(* Logix 5000 project; controller CLASE_1 Emulate 5570 rev 28.11; software revision 28.02; part 9 of 15 *)
(* tags used below, declared in another part *)
   Inp_ActuatorFault : BOOL;   // Valve Actuator Fault (overload, etc.), 0=OK, 1=Fault)
   Cfg_SetTrack : BOOL;   // 1=PSets track OSets in Oper, OSets track PSets in Prog, 0=no tracking
   Cfg_SetTrackOvrdHand : BOOL;   // 1=Prog/Oper Settings track Override/Hand CV
   Cfg_MinCV : REAL;   // Minimum CV (in CV EU, for limiting)
   Cfg_MaxCV : REAL;   // Maximum CV (in CV EU, for limiting)
   Cfg_CycleT : REAL;   // Open and Close Pulse Output overall period (s)
   Cfg_OpenRate : REAL;   // Rate at which valve moves when opening (CV EU/sec)
   Cfg_CloseRate : REAL;   // Rate at which valve moves when closing (CV EU/sec)
   Cfg_MaxOnT : REAL;   // Open and Close Pulse Output maximum ON time (s)
   Cfg_MinOnT : REAL;   // Open and Close Pulse Output minimum ON time (s)
   Cfg_BumpT : REAL;   // Time to bump valve open or closed (by Oper) when Fdbk Bad (sec)
   Cfg_Deadtime : REAL;   // Additional time on first pulse after stop or direction change
   PSet_CV : REAL;   // Program Setting of Controlled Variable (output) (CV EU)
   PSet_CVRoCLimInc : REAL;   // Program Setting of CV Rate of Change Limit, Increasing, (in EU/sec)
   PSet_CVRoCLimDec : REAL;   // Program Setting of CV Rate of Change Limit, Decreasing, (in EU/sec)
   OSet_CV : REAL;   // Operator Setting of Controlled Variable (output) (CV EU)
   OSet_CVRoCLimInc : REAL;   // Operator Setting of CV Rate of Change Limit, Increasing, (in EU/sec)
   OSet_CVRoCLimDec : REAL;   // Operator Setting of CV Rate of Change Limit, Decreasing, (in EU/sec)
   Out_Open : BOOL;   // Pulse Output to drive valve Open
   Out_Close : BOOL;   // Pulse Output to drive valve closed
   Val_Pos : REAL;   // Valve actual position from feedback (CV EU)
   Val_CVSet : REAL;   // Value of selected CV Setting (before rate limiting, CV EU)
   Val_CVOut : REAL;   // Value of CV output (after clamping and ramping) (CV EU)
   Val_CVRoCLimInc : REAL;   // Value of CV Rate of Change Limit, Increasing, (in EU/sec)
   Val_CVRoCLimDec : REAL;   // Value of CV Rate of Change Limit, Decreasing, (in EU/sec)
   Sts_BumpOpen : BOOL;   // 1=Bump Open Requested or Active
   Sts_BumpClose : BOOL;   // 1=Bump Close Requested or Active
   Sts_Ramping : BOOL;   // 1=CV is ramping to target
   Sts_Clamped : BOOL;   // 1=CV Set is clamped at CVMin or CVMax
   P_ValveC : BOOL;   // Unique Parameter Name for auto - discovery
   Wrk_CVRoCLimInc : REAL;   // Selected CV Rate of Change Limit Increasing
   Wrk_CVSet : REAL;   // Final selected CV to feed to RoC Limiter
   Wrk_CVOut : REAL;   // Working value of CV after Rate Limiting
   ActuatorFault : P_Alarm;   // Actuator Fault Alarm (based on Actuator Fault Input)
   Wrk_Close : BOOL;   // Internal Close output -- before Sim
   Wrk_CycleT : TIMER;   // Overall Cycle Timer for pulsed outputs
   Wrk_OKtoOpen : BOOL;   // OK to pulse Out_Open
   Wrk_OKtoClose : BOOL;   // OK to pulse Out_Close
   Wrk_OpenTime : REAL;   // Time to pulse Out_Open
   Wrk_CycleT_ms : DINT;   // Cycle Time in milliseconds (preset)
   Wrk_OpenTimePrev : DINT;   // Wrk_OpenTime from previous cycle
   Wrk_CloseTime : REAL;   // Time to pulse Out_Close
   Wrk_CloseTimePrev : REAL;   // Wrk_CloseTime from previous cycle
   Wrk_CVRoCLimDec : REAL;   // Selected CV Rate of Change Limit Decreasing
   Wrk_BumpClose : BOOL;   // Operator Bump Close requested
   Wrk_BumpOpen : BOOL;   // Operator Bump Open requested
   Wrk_BumpingOpen : BOOL;   // Operator Bump Open actively pulsing Out_Open
   Wrk_BumpingClose : BOOL;   // Operator Bump Close actively pulsing Out_Close
   Wrk_CycleActive : BOOL;   // Outputs are cycling; wait for cycle to complete
   Wrk_ShedIntlkCV : BOOL;   // Output CV being held at Interlock value
   Wrk_ShedHold : BOOL;   // Output CV being held at last good value
(* P_ValveC, continued *)

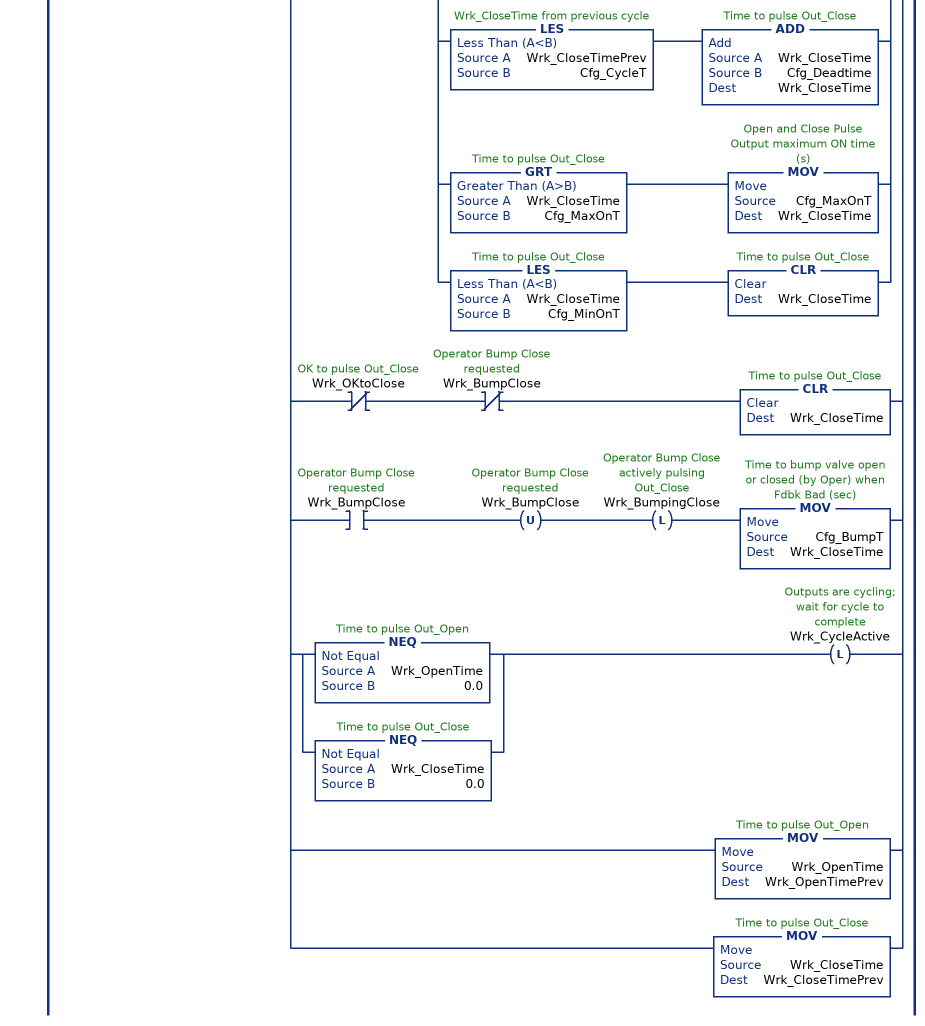
   // When the Cycle completes, calculate a new Open Time (time to pulse the
   // Open output) and Close Time (time to pulse the Close output).
   // Details of this calculation are in the Instruction Help for the POSP built-in
   // instruction, from which this logic is derived.
   48: [GEQ(Wrk_CycleT.ACC,Wrk_CycleT_ms) ,XIO(Wrk_CycleActive) ][OTU(Wrk_CycleActive) OTU(Wrk_BumpingOpen) OTU(Wrk_BumpingClose) CLR(Wrk_CycleT.ACC) ,XIC(Wrk_OKtoOpen) [CPT(Wrk_OpenTime,(Val_CVOut-Val_Pos)/Cfg_OpenRate) ,LES(Wrk_OpenTimePrev,Cfg_CycleT) ADD(Wrk_OpenTime,Cfg_Deadtime,Wrk_OpenTime) ,GRT(Wrk_OpenTime,Cfg_MaxOnT) MOV(Cfg_MaxOnT,Wrk_OpenTime) ,LES(Wrk_OpenTime,Cfg_MinOnT) CLR(Wrk_OpenTime) ] ,XIO(Wrk_OKtoOpen) XIO(Wrk_BumpOpen) CLR(Wrk_OpenTime) ,XIC(Wrk_BumpOpen) OTU(Wrk_BumpOpen) OTL(Wrk_BumpingOpen) MOV(Cfg_BumpT,Wrk_OpenTime) ,XIC(Wrk_OKtoClose) [CPT(Wrk_CloseTime,(Val_Pos-Val_CVOut)/Cfg_CloseRate) ,LES(Wrk_CloseTimePrev,Cfg_CycleT) ADD(Wrk_CloseTime,Cfg_Deadtime,Wrk_CloseTime) ,GRT(Wrk_CloseTime,Cfg_MaxOnT) MOV(Cfg_MaxOnT,Wrk_CloseTime) ,LES(Wrk_CloseTime,Cfg_MinOnT) CLR(Wrk_CloseTime) ] ,XIO(Wrk_OKtoClose) XIO(Wrk_BumpClose) CLR(Wrk_CloseTime) ,XIC(Wrk_BumpClose) OTU(Wrk_BumpClose) OTL(Wrk_BumpingClose) MOV(Cfg_BumpT,Wrk_CloseTime) ,[NEQ(Wrk_OpenTime,0.0) ,NEQ(Wrk_CloseTime,0.0) ] OTL(Wrk_CycleActive) ,MOV(Wrk_OpenTime,Wrk_OpenTimePrev) ,MOV(Wrk_CloseTime,Wrk_CloseTimePrev) ];
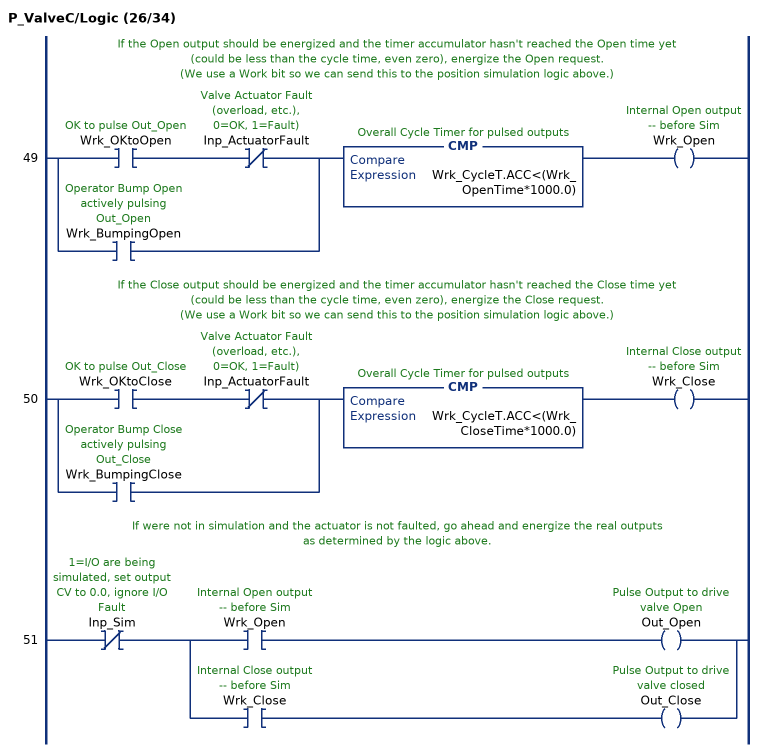
   // If the Open output should be energized and the timer accumulator hasn't reached the Open time yet
   // (could be less than the cycle time, even zero), energize the Open request.
   // (We use a Work bit so we can send this to the position simulation logic above.)
   49: [XIC(Wrk_OKtoOpen) XIO(Inp_ActuatorFault) ,XIC(Wrk_BumpingOpen) ]CMP(Wrk_CycleT.ACC<(Wrk_OpenTime*1000.0))OTE(Wrk_Open);
   // If the Close output should be energized and the timer accumulator hasn't reached the Close time yet
   // (could be less than the cycle time, even zero), energize the Close request.
   // (We use a Work bit so we can send this to the position simulation logic above.)
   50: [XIC(Wrk_OKtoClose) XIO(Inp_ActuatorFault) ,XIC(Wrk_BumpingClose) ]CMP(Wrk_CycleT.ACC<(Wrk_CloseTime*1000.0))OTE(Wrk_Close);
   // If were not in simulation and the actuator is not faulted, go ahead and energize the real outputs
   // as determined by the logic above.
   51: XIO(Inp_Sim)[XIC(Wrk_Open) OTE(Out_Open) ,XIC(Wrk_Close) OTE(Out_Close) ];
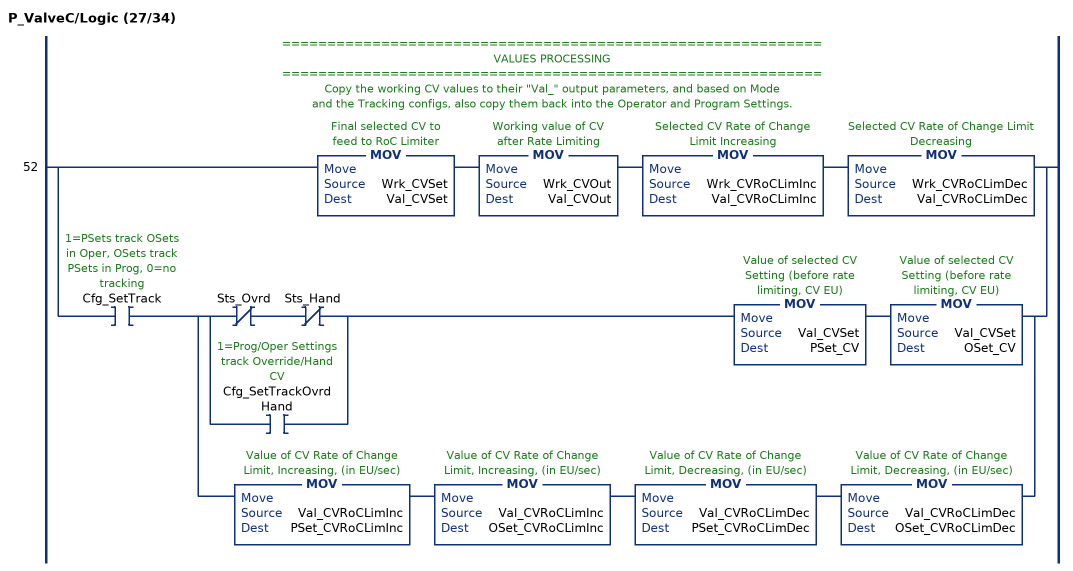
   // ============================================================
   // VALUES PROCESSING
   // ============================================================
   // Copy the working CV values to their "Val_" output parameters, and based on Mode
   // and the Tracking configs, also copy them back into the Operator and Program Settings.
   52: [MOV(Wrk_CVSet,Val_CVSet) MOV(Wrk_CVOut,Val_CVOut) MOV(Wrk_CVRoCLimInc,Val_CVRoCLimInc) MOV(Wrk_CVRoCLimDec,Val_CVRoCLimDec) ,XIC(Cfg_SetTrack) [[XIO(Sts_Ovrd) XIO(Sts_Hand) ,XIC(Cfg_SetTrackOvrdHand) ] MOV(Val_CVSet,PSet_CV) MOV(Val_CVSet,OSet_CV) ,MOV(Val_CVRoCLimInc,PSet_CVRoCLimInc) MOV(Val_CVRoCLimInc,OSet_CVRoCLimInc) MOV(Val_CVRoCLimDec,PSet_CVRoCLimDec) MOV(Val_CVRoCLimDec,OSet_CVRoCLimDec) ] ];
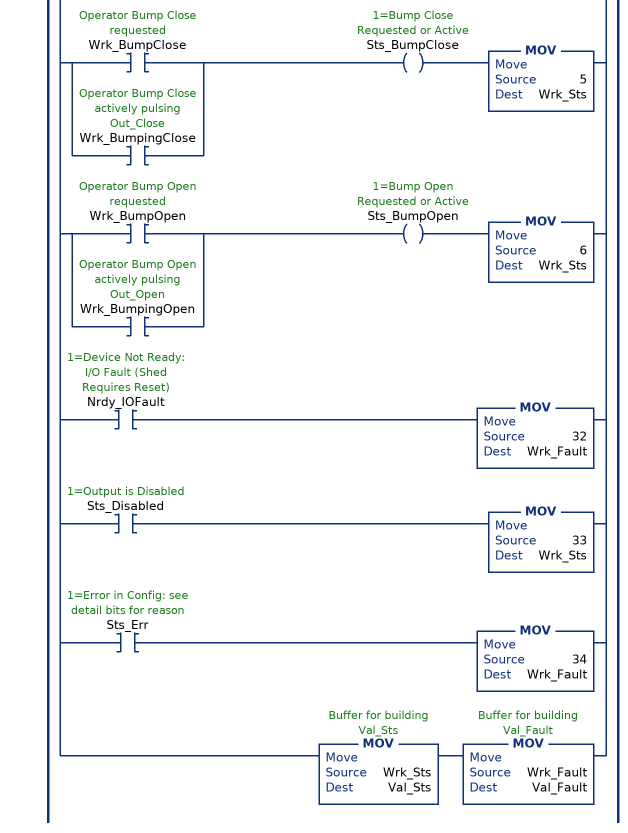
   // Val_Sts is the current device status, as determined by this AOI,
   // based on its knowledge of settings and configuration.
   // (This is the status that should be monitored by, for example, FT Historian.)
   // 0 = At Target
   // 1 = Ramping Down
   // 2 = Ramping Up
   // 3 = Clamped at CVMin
   // 4 = Clamped at CVMax
   // 5 = Bump Close requested or currently pulsing Out_Close
   // 6 = Bump Open requested or currently pulsing Out_Open
   // 32 = I/O Fault
   // 33 = Disabled
   // 34 = Configuration Error
   // #####  V3.0-04  2014-01-20:  Corrected generation of Val_Sts, Val_Fault.  #####
   // #####  V3.1-00  2014-07-22: Added Not Ready reason bits (Nrdy_xxx)  #####
   // #####  V3.1-03  2015-01-21:  Modified to show Val_Sts = 1 or 2 when moving via pulsing.  #####
   53: [CLR(Wrk_Sts) CLR(Wrk_Fault) ,[GRT(Wrk_OpenTime,0.0) XIO(Inp_ActuatorFault) ,XIC(Sts_Ramping) LES(Wrk_CVOut,Wrk_CVSet) ] MOV(2,Wrk_Sts) ,[GRT(Wrk_CloseTime,0.0) XIO(Inp_ActuatorFault) ,XIC(Sts_Ramping) GRT(Wrk_CVOut,Wrk_CVSet) ] MOV(1,Wrk_Sts) ,XIC(Sts_Clamped) [EQU(Wrk_CVOut,Cfg_MinCV) MOV(3,Wrk_Sts) ,EQU(Wrk_CVOut,Cfg_MaxCV) MOV(4,Wrk_Sts) ] ,[XIC(Wrk_BumpClose) ,XIC(Wrk_BumpingClose) ] OTE(Sts_BumpClose) MOV(5,Wrk_Sts) ,[XIC(Wrk_BumpOpen) ,XIC(Wrk_BumpingOpen) ] OTE(Sts_BumpOpen) MOV(6,Wrk_Sts) ,XIC(Nrdy_IOFault) MOV(32,Wrk_Fault) ,XIC(Sts_Disabled) MOV(33,Wrk_Sts) ,XIC(Sts_Err) MOV(34,Wrk_Fault) ,MOV(Wrk_Sts,Val_Sts) MOV(Wrk_Fault,Val_Fault) ];
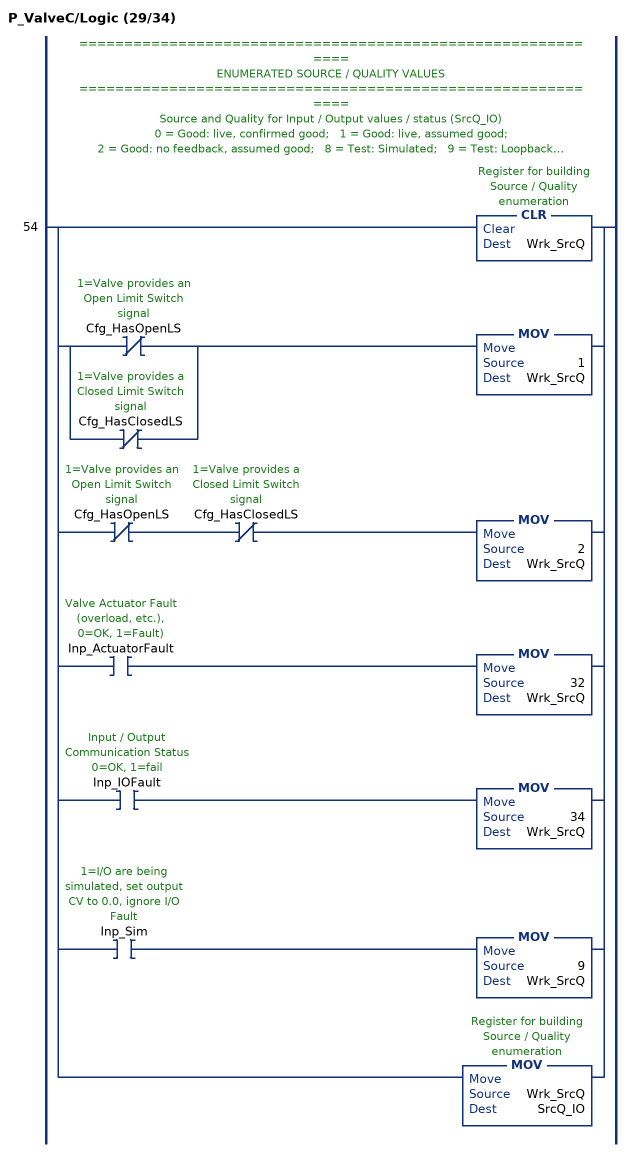
   // ============================================================
   // ENUMERATED SOURCE / QUALITY VALUES
   // ============================================================
   // Source and Quality for Input / Output values / status (SrcQ_IO)
   // 0 = Good: live, confirmed good;   1 = Good: live, assumed good;
   // 2 = Good: no feedback, assumed good;   8 = Test: Simulated;   9 = Test: Loopback;
   // 10 = Test: Manually Entered;   16 = Uncertain: Live, off-spec;
   // 17 = Uncertain, Substituted at Device / Bus;   18 = Uncertain, Substituted at AOI;
   // 19 = Uncertain, using last known good;    20 = Uncertain, using replacement value;
   // 32 = Bad, Signal Failure;   33 = Bad, Channel Fault;
   // 34 = Bad, Module / Comms Fault;   35 = Bad, Invalid Configuration
   // #####  V3.1-00  2014-07-22:  Added rung for Source/Quality enumerations.  #####
   54: [CLR(Wrk_SrcQ) ,[XIO(Cfg_HasOpenLS) ,XIO(Cfg_HasClosedLS) ] MOV(1,Wrk_SrcQ) ,XIO(Cfg_HasOpenLS) XIO(Cfg_HasClosedLS) MOV(2,Wrk_SrcQ) ,XIC(Inp_ActuatorFault) MOV(32,Wrk_SrcQ) ,XIC(Inp_IOFault) MOV(34,Wrk_SrcQ) ,XIC(Inp_Sim) MOV(9,Wrk_SrcQ) ,MOV(Wrk_SrcQ,SrcQ_IO) ];
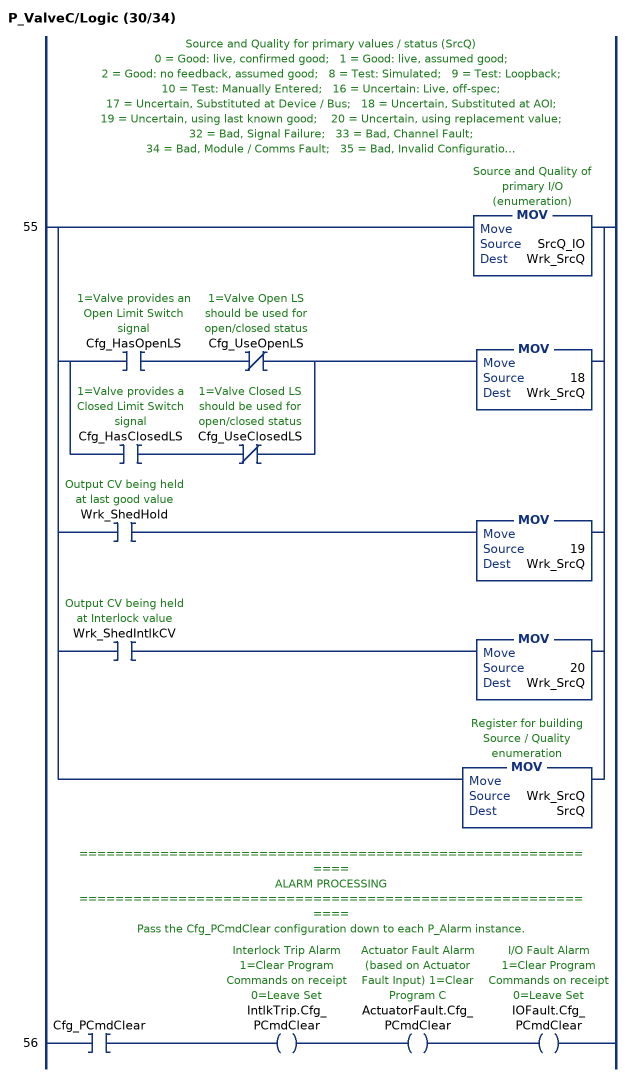
   // Source and Quality for primary values / status (SrcQ)
   // 0 = Good: live, confirmed good;   1 = Good: live, assumed good;
   // 2 = Good: no feedback, assumed good;   8 = Test: Simulated;   9 = Test: Loopback;
   // 10 = Test: Manually Entered;   16 = Uncertain: Live, off-spec;
   // 17 = Uncertain, Substituted at Device / Bus;   18 = Uncertain, Substituted at AOI;
   // 19 = Uncertain, using last known good;    20 = Uncertain, using replacement value;
   // 32 = Bad, Signal Failure;   33 = Bad, Channel Fault;
   // 34 = Bad, Module / Comms Fault;   35 = Bad, Invalid Configuration
   // #####  V3.1-00  2014-07-22:  Added rung for Source/Quality enumerations.  #####
   55: [MOV(SrcQ_IO,Wrk_SrcQ) ,[XIC(Cfg_HasOpenLS) XIO(Cfg_UseOpenLS) ,XIC(Cfg_HasClosedLS) XIO(Cfg_UseClosedLS) ] MOV(18,Wrk_SrcQ) ,XIC(Wrk_ShedHold) MOV(19,Wrk_SrcQ) ,XIC(Wrk_ShedIntlkCV) MOV(20,Wrk_SrcQ) ,MOV(Wrk_SrcQ,SrcQ) ];
   // ============================================================
   // ALARM PROCESSING
   // ============================================================
   // Pass the Cfg_PCmdClear configuration down to each P_Alarm instance.
   56: XIC(Cfg_PCmdClear)OTE(IntlkTrip.Cfg_PCmdClear)OTE(ActuatorFault.Cfg_PCmdClear)OTE(IOFault.Cfg_PCmdClear);
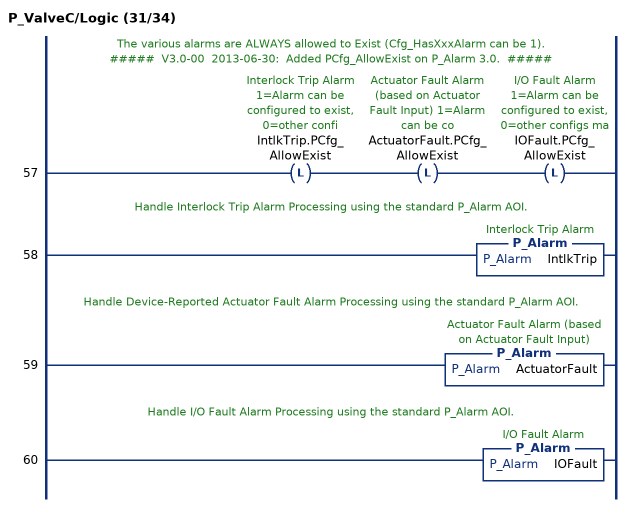
   // The various alarms are ALWAYS allowed to Exist (Cfg_HasXxxAlarm can be 1).
   // #####  V3.0-00  2013-06-30:  Added PCfg_AllowExist on P_Alarm 3.0.  #####
   57: OTL(IntlkTrip.PCfg_AllowExist)OTL(ActuatorFault.PCfg_AllowExist)OTL(IOFault.PCfg_AllowExist);
   // Handle Interlock Trip Alarm Processing using the standard P_Alarm AOI.
   58: P_Alarm(IntlkTrip);
   // Handle Device-Reported Actuator Fault Alarm Processing using the standard P_Alarm AOI.
   59: P_Alarm(ActuatorFault);
   // Handle I/O Fault Alarm Processing using the standard P_Alarm AOI.
   60: P_Alarm(IOFault);
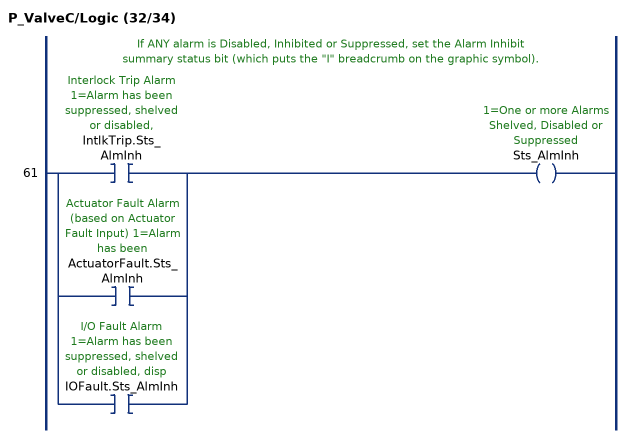
   // If ANY alarm is Disabled, Inhibited or Suppressed, set the Alarm Inhibit
   // summary status bit (which puts the "I" breadcrumb on the graphic symbol).
   61: [XIC(IntlkTrip.Sts_AlmInh) ,XIC(ActuatorFault.Sts_AlmInh) ,XIC(IOFault.Sts_AlmInh) ]OTE(Sts_AlmInh);
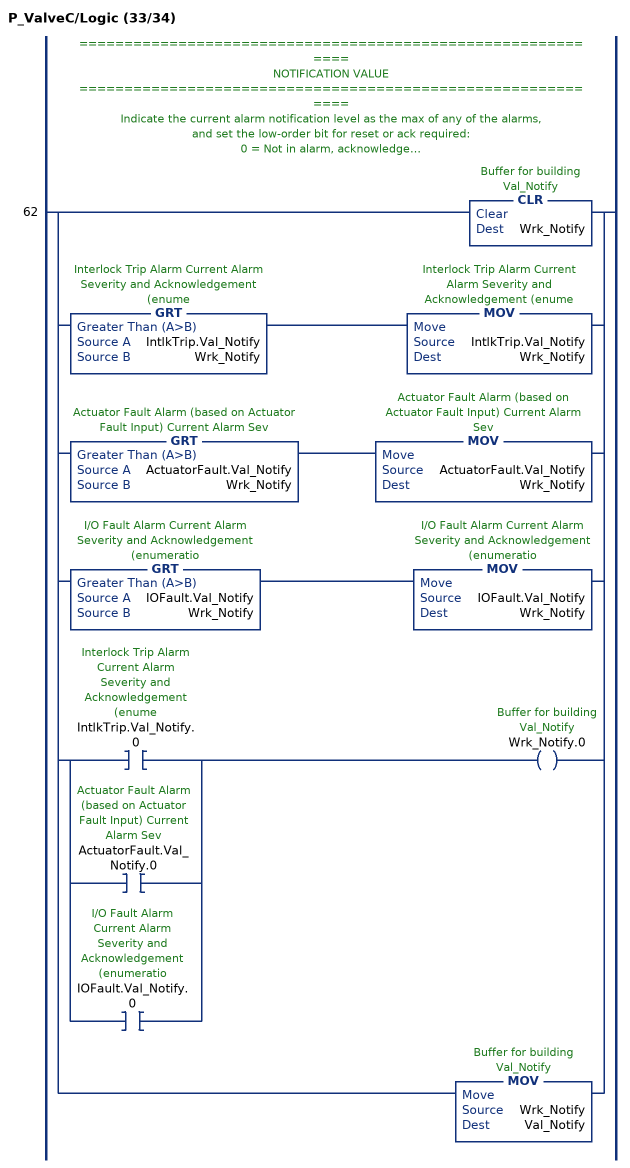
   // ============================================================
   // NOTIFICATION VALUE
   // ============================================================
   // Indicate the current alarm notification level as the max of any of the alarms,
   // and set the low-order bit for reset or ack required:
   // 0 = Not in alarm, acknowledged
   // 1 = Not in alarm, unacknowledged or reset required
   // 2 = Low severity alarm, acknowledged
   // 3 = Low severity alarm, unacknowledged
   // 4 = Medium severity alarm, acknowledged
   // 5 = Medium severity alarm, unacknowledged
   // 6 = High severity alarm, acknowledged
   // 7 = High severity alarm, unacknowledged
   // 8 = Urgent severity alarm, acknowledged
   // 9 = Urgent severity alarm, unacknowledged
   // #####  V3.1-00  2014-07-22:  Separated Reset Reqd functions from Val_Notify  #####
   62: [CLR(Wrk_Notify) ,GRT(IntlkTrip.Val_Notify,Wrk_Notify) MOV(IntlkTrip.Val_Notify,Wrk_Notify) ,GRT(ActuatorFault.Val_Notify,Wrk_Notify) MOV(ActuatorFault.Val_Notify,Wrk_Notify) ,GRT(IOFault.Val_Notify,Wrk_Notify) MOV(IOFault.Val_Notify,Wrk_Notify) ,[XIC(IntlkTrip.Val_Notify.0) ,XIC(ActuatorFault.Val_Notify.0) ,XIC(IOFault.Val_Notify.0) ] OTE(Wrk_Notify.0) ,MOV(Wrk_Notify,Val_Notify) ];
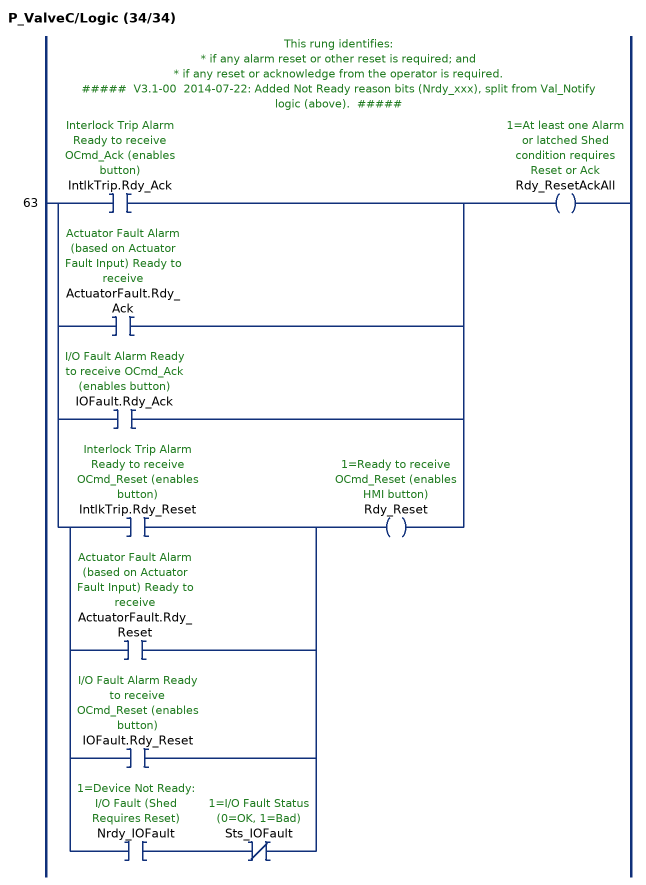
   // This rung identifies:
   // * if any alarm reset or other reset is required; and
   // * if any reset or acknowledge from the operator is required.
   // #####  V3.1-00  2014-07-22: Added Not Ready reason bits (Nrdy_xxx), split from Val_Notify logic (above).  #####
   63: [[XIC(IntlkTrip.Rdy_Ack) ,XIC(ActuatorFault.Rdy_Ack) ,XIC(IOFault.Rdy_Ack) ] ,[XIC(IntlkTrip.Rdy_Reset) ,XIC(ActuatorFault.Rdy_Reset) ,XIC(IOFault.Rdy_Reset) ,XIC(Nrdy_IOFault) XIO(Sts_IOFault) ] OTE(Rdy_Reset) ]OTE(Rdy_ResetAckAll);
END_ROUTINE

ROUTINE Prescan   (* ladder *)
// Clear Ownership. clear "lurking" Commands
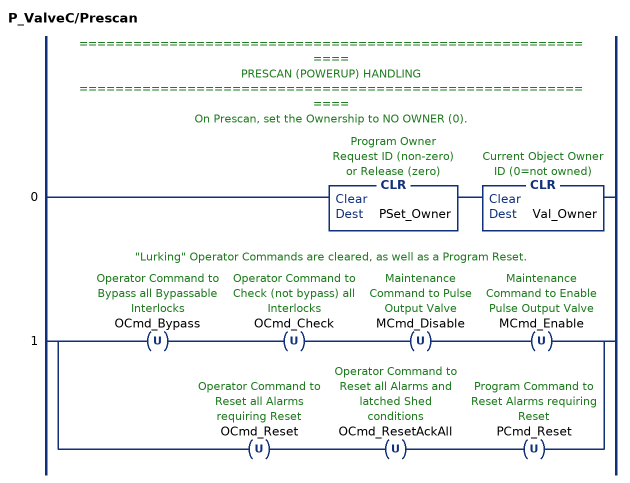
   // ============================================================
   // PRESCAN (POWERUP) HANDLING
   // ============================================================
   // On Prescan, set the Ownership to NO OWNER (0).
   0: CLR(PSet_Owner)CLR(Val_Owner);
   // "Lurking" Operator Commands are cleared, as well as a Program Reset.
   1: [OTU(OCmd_Bypass) OTU(OCmd_Check) OTU(MCmd_Disable) OTU(MCmd_Enable) ,OTU(OCmd_Reset) OTU(OCmd_ResetAckAll) OTU(PCmd_Reset) ];
END_ROUTINE
END_ADD_ON_INSTRUCTION

ADD_ON_INSTRUCTION P_ValveSO   (* revision 3.5 04 Release, vendor Rockwell Automation, ExecutePrescan, ExecuteEnableInFalse *)
// Solenoid Operated Valve
// Revision note:
// See V3.5-xx Release Notes for details. Modified to align
// with actual device state on transition from Sim to real valve.
// Help:
// Copyright © Rockwell Automation, Inc.  All Rights Reserved.
// This Instruction controls and monitors a single solenoid operated
// valve (two position: opened, closed) and provides:
// *  Support for fail open (energize to close) and fail closed (energize to open, default) valves
// *  Monitoring of limit switch feedback, display of actual valve status
// *  Detection of Failure to Open, Failure to Close
// *  Monitoring of Permissive conditions to allow energizing
// *  Monitoring of Interlock conditions to de-energize
// *  Simulation, providing feedback of a working valve while disabling outputs
// *  Monitoring of I/O communication faults
// *  Alarms for Full Stall (didn't move), Transit Stall (didn't reach target position), Interlock Trip, I/O Fault
// *  Operation in Hand, Maintenance, Override, Program and Operator Modes
// *  "Available" status for use by automation logic to know whether valve
//       can be controlled by other objects.
// Modes are provided by a P_Mode AOI instance.
// Alarms are provided by P_Alarm AOI instances.
// Modes of operation: Operator, Program, Override, Maintenance, Hand
VAR_INPUT
   Inp_OpenLS : BOOL; {visible}   // Valve Open Limit Switch 1=confirmed OPEN
   Inp_ClosedLS : BOOL; {visible}   // Valve Closed Limit Switch 1=confirmed CLOSED
   Inp_PermOK : BOOL := 1; {visible}   // 1=Permissives OK, Valve can energize
   Inp_NBPermOK : BOOL := 1; {visible}   // 1=Non-Bypassable Permissives OK, valve can energize
   Inp_IntlkOK : BOOL := 1; {visible}   // 1=Interlocks OK, valve can energize
   Inp_NBIntlkOK : BOOL := 1; {visible}   // 1=Non-Bypassable Interlocks OK, valve can energize
   Inp_IOFault : BOOL;   // Input Communication Status 0=OK, 1=fail
   Inp_Sim : BOOL;   // 1=Simulate working valve; 0=Open/Close/ Monitor actual valve
   Inp_Hand : ALIAS FOR Mode.Inp_Hand; {visible}
   Inp_Ovrd : ALIAS FOR Mode.Inp_Ovrd; {visible}
   Inp_OvrdCmd : DINT; {visible}   // Override Mode Command: 0=None, 1=Close, 2=Open
   Inp_Reset : BOOL; {visible}   // 1=Reset all fault conditions and latched Alarms
   Cfg_FailOpen : BOOL;   // 1=Fail Open (energize to close), 0=Fail Closed (energize to open)
   Cfg_HasOpenLS : BOOL;   // 1=Valve provides an Open Limit Switch signal
   Cfg_HasClosedLS : BOOL;   // 1=Valve provides a Closed Limit Switch signal
   Cfg_UseOpenLS : BOOL;   // 1=Valve Open LS should be used for failure checking
   Cfg_UseClosedLS : BOOL;   // 1=Valve Closed LS should be used for failure checking
   Cfg_LSFail : BOOL := 1;   // 1=both switches ON=fail, 0=both switches OFF=fail
   Cfg_HasPermObj : BOOL;   // 1=Tells HMI a P_Perm is connected to Inp_Perm
   Cfg_HasIntlkObj : BOOL;   // 1=Tells HMI a P_Intlk is connected to Inp_Intlk
   Cfg_HasStatsObj : BOOL;   // 1=Tells HMI a P_ValveStats is monitoring this valve
   Cfg_PCmdClear : ALIAS FOR Mode.Cfg_PCmdClear;
   Cfg_ProgDefault : ALIAS FOR Mode.Cfg_ProgDefault;
   Cfg_OCmdResets : BOOL;   // 1=New Oper valve cmd. resets fault, 0=reset req'd to clear fault
   Cfg_ShedOnFullStall : BOOL := 1;   // 1=Stop Valve and Alarm on Full Stall; 0=Alarm only on Full Stall
   Cfg_ShedOnTransitStall : BOOL := 1;   // 1=Stop Valve and Alarm on Transit Stall; 0=Alarm only on Transit Stall
   Cfg_ShedOnIOFault : BOOL := 1;   // 1=Stop Valve and Alarm on I/O Fault; 0=Alarm only on I/O Fault
   Cfg_OvrdPermIntlk : BOOL;   // 1=Override ignores Bypassable Perm/ Intlk; 0=always use Perm/Intlk
   Cfg_HasFullStallAlm : ALIAS FOR FullStall.Cfg_Exists;   // 1=Full Stall Alarm exists and will be checked
   Cfg_HasTransitStallAlm : ALIAS FOR TransitStall.Cfg_Exists;   // 1=Transit Stall Alarm exists and will be checked
   Cfg_HasIntlkTripAlm : ALIAS FOR IntlkTrip.Cfg_Exists;   // 1=Interlock Trip Alarm exists and will be checked
   Cfg_HasIOFaultAlm : ALIAS FOR IOFault.Cfg_Exists;   // 1=I/O Fault Alarm exists and will be checked
   Cfg_FullStallResetReqd : ALIAS FOR FullStall.Cfg_ResetReqd;   // 1=Reset requied to clear Full Stall Alarm
   Cfg_TransitStallResetReqd : ALIAS FOR TransitStall.Cfg_ResetReqd;   // 1=Reset required to clear Transit Stall Alarm
   Cfg_IntlkTripResetReqd : ALIAS FOR IntlkTrip.Cfg_ResetReqd;   // 1=Reset required to clear Interlock Trip Alarm
   Cfg_IOFaultResetReqd : ALIAS FOR IOFault.Cfg_ResetReqd;   // 1=Reset required to clear I/O Fault Alarm
   Cfg_FullStallAckReqd : ALIAS FOR FullStall.Cfg_AckReqd;   // 1=Acknowledge required for Full Stall Alarm
   Cfg_TransitStallAckReqd : ALIAS FOR TransitStall.Cfg_AckReqd;   // 1=Acknowledge required for Transit Stall Alarm
   Cfg_IntlkTripAckReqd : ALIAS FOR IntlkTrip.Cfg_AckReqd;   // 1=Acknowledge required for Interlock Trip Alarm
   Cfg_IOFaultAckReqd : ALIAS FOR IOFault.Cfg_AckReqd;   // 1=Acknowledge required for I/O Fault Alarm
   Cfg_FullStallSeverity : ALIAS FOR FullStall.Cfg_Severity;   // Full Stall Alarm Severity: 1..250=Low, 251..500=Medium, 501..750=High, 751..1000=Urgent
   Cfg_TransitStallSeverity : ALIAS FOR TransitStall.Cfg_Severity;   // Transit Stall Alarm Severity: 1..250=Low, 251..500=Medium, 501..750=High, 751..1000=Urgent
   Cfg_IntlkTripSeverity : ALIAS FOR IntlkTrip.Cfg_Severity;   // Interlock Trip Alarm Severity: 1..250=Low, 251..500=Medium, 501..750=High, 751..1000=Urgent
   Cfg_IOFaultSeverity : ALIAS FOR IOFault.Cfg_Severity;   // I/O Fault Alarm Severity: 1..250=Low, 251..500=Medium, 501..750=High, 751..1000=Urgent
   Cfg_SimFdbkT : DINT := 2;   // Delay to echo back of Open/Closed status when in Simulation (sec)
   Cfg_FullStallT : DINT := 5;   // After command, time with no motion before Fault (sec)
   Cfg_TransitStallT : DINT := 10;   // After command, time to reach position before fault (sec)
   PSet_Owner : DINT;   // Program Owner Request ID (non-zero) or Release (zero)
   PCmd_Open : BOOL;   // Program Command to Open Valve
   PCmd_Close : BOOL;   // Program Command to Close Valve
   PCmd_Acq : ALIAS FOR Mode.PCmd_Acq;
   PCmd_Rel : ALIAS FOR Mode.PCmd_Rel;
   PCmd_Lock : ALIAS FOR Mode.PCmd_Lock;
   PCmd_Unlock : ALIAS FOR Mode.PCmd_Unlock;
   PCmd_Reset : BOOL;   // Program Command to Reset all Alarms requiring Reset
   PCmd_FullStallAck : ALIAS FOR FullStall.PCmd_Ack;   // Program Command to Acknowledge Full Stall Alarm
   PCmd_FullStallSuppress : ALIAS FOR FullStall.PCmd_Suppress;   // Program Command to Suppress Full Stall Alarm
   PCmd_FullStallUnsuppress : ALIAS FOR FullStall.PCmd_Unsuppress;   // Program Command to Unsuppress Full Stall Alarm
   PCmd_FullStallUnshelve : ALIAS FOR FullStall.PCmd_Unshelve;   // Program Command to Unshelve Full Stall Alarm
   PCmd_TransitStallAck : ALIAS FOR TransitStall.PCmd_Ack;   // Program Command to Acknowledge Transit Stall Alarm
   PCmd_TransitStallSuppress : ALIAS FOR TransitStall.PCmd_Suppress;   // Program Command to Suppress Transit Stall Alarm
   PCmd_TransitStallUnsuppress : ALIAS FOR TransitStall.PCmd_Unsuppress;   // Program Command to Unsuppress Transit Stall Alarm
   PCmd_TransitStallUnshelve : ALIAS FOR TransitStall.PCmd_Unshelve;   // Program Command to Unshelve Transit Stall Alarm
   PCmd_IntlkTripAck : ALIAS FOR IntlkTrip.PCmd_Ack;   // Program Command to Acknowledge Interlock Trip Alarm
   PCmd_IntlkTripSuppress : ALIAS FOR IntlkTrip.PCmd_Suppress;   // Program Command to Suppress Interlock Trip Alarm
   PCmd_IntlkTripUnsuppress : ALIAS FOR IntlkTrip.PCmd_Unsuppress;   // Program Command to Unsuppress Interlock Trip Alarm
   PCmd_IntlkTripUnshelve : ALIAS FOR IntlkTrip.PCmd_Unshelve;   // Program Command to Unshelve Interlock Trip Alarm
   PCmd_IOFaultAck : ALIAS FOR IOFault.PCmd_Ack;   // Program Command to Acknowledge I/O Fault Alarm
   PCmd_IOFaultSuppress : ALIAS FOR IOFault.PCmd_Suppress;   // Program Command to Suppress I/O Fault Alarm
   PCmd_IOFaultUnsuppress : ALIAS FOR IOFault.PCmd_Unsuppress;   // Program Command to Unsuppress I/O Fault Alarm
   PCmd_IOFaultUnshelve : ALIAS FOR IOFault.PCmd_Unshelve;   // Program Command to Unshelve I/O Fault Alarm
   OCmd_Open : BOOL;   // Operator Command to Open Valve
   OCmd_Close : BOOL;   // Operator Command to Close Valve
   OCmd_Bypass : BOOL;   // Operator Command to Bypass all Bypassable Interlocks and Permissives
   OCmd_Check : BOOL;   // Operator Command to Check (not bypass) all Interlocks and Permissives
   MCmd_Disable : BOOL;   // Maintenance Command to Disable Valve
   MCmd_Enable : BOOL;   // Maintenance Command to Enable (allow to energize) Valve
   MCmd_Acq : ALIAS FOR Mode.MCmd_Acq;
   MCmd_Rel : ALIAS FOR Mode.MCmd_Rel;
   OCmd_AcqLock : ALIAS FOR Mode.OCmd_AcqLock;
   OCmd_Unlock : ALIAS FOR Mode.OCmd_UnlockRel;
   OCmd_Reset : BOOL;   // Operator Command to Reset all Alarms requiring Reset
   OCmd_ResetAckAll : BOOL;   // Operator Command to Reset all Alarms and latched Shed conditions
END_VAR
VAR_OUTPUT
   Out : BOOL; {access Read Only, visible}   // 1=Energize Valve Solenoid
   SrcQ_IO : SINT; {access Read Only}   // Source and Quality of primary I/O (enumeration)
   SrcQ : SINT; {access Read Only}   // Source and Quality of primary Val/Sts (enumeration)
   Val_Cmd : SINT; {access Read Only}   // Device Command 0=None, 1=Close, 2=Open
   Val_Fdbk : SINT; {access Read Only}   // Device Feedback 0=Moving, 1=Closed, 2=Opened, 3=Limit Switch Failure
   Val_Sts : SINT; {access Read Only}   // Device Confirmed Sts 0=? 1=Closed 2=Open 5=Closing, 6=Opening, 33=Disabled
   Val_Fault : SINT; {access Read Only}   // Device Fault Status 0=None, 16=Transit Stall, 17 = Full Stall, 32=I/O Fault, 34=Config Error
   Val_Mode : ALIAS FOR Mode.Val; {access Read Only}
   Val_Owner : DINT; {access Read Only}   // Current Object Owner ID (0=not owned)
   Val_Notify : SINT; {access Read Only}   // Current Alarm Level and Acknowledgement (enumeration)
   Sts_Closed : BOOL; {access Read Only, visible}   // 1=Valve requested to Close and is confirmed Closed
   Sts_Opening : BOOL; {access Read Only, visible}   // 1=Valve requested to open and awaiting open feedback
   Sts_Opened : BOOL; {access Read Only, visible}   // 1=Valve requested to open and is confirmed Opened
   Sts_Closing : BOOL; {access Read Only, visible}   // 1=Valve requested to Close and awaiting Closed feedback
   Sts_Available : BOOL; {access Read Only}   // 1=Valve available for control by automation (Prog)
   Sts_Bypass : BOOL; {access Read Only}   // 1=Bypassable Interlocks and Permissives are Bypassed
   Sts_BypActive : BOOL; {access Read Only}   // 1=Bypassing Active (Bypassed or Maintenance)
   Sts_Disabled : BOOL; {access Read Only}   // 1=Valve is Disabled
   Sts_LSFail : BOOL; {access Read Only}   // 1=Limit Switch Overlap Failure
   Sts_NotRdy : BOOL; {access Read Only}   // 1=Device Not Ready, see detail bits for reason
   Nrdy_Disabled : BOOL; {access Read Only}   // 1=Device Not Ready: Device Disabled by Maintenance
   Nrdy_CfgErr : BOOL; {access Read Only}   // 1=Device Not Ready: Configuration Error
   Nrdy_Intlk : BOOL; {access Read Only}   // 1=Device Not Ready: Interlock Not OK
   Nrdy_Perm : BOOL; {access Read Only}   // 1=Device Not Ready: Permissive Not OK
   Nrdy_Fail : BOOL; {access Read Only}   // 1=Device Not Ready: Device Failure (Shed Requires Reset)
   Nrdy_IOFault : BOOL; {access Read Only}   // 1=Device Not Ready: I/O Fault (Shed Requires Reset)
   Nrdy_NoMode : BOOL; {access Read Only}   // 1=Device Not Ready: Device Logic Disabled / NO Mode
   Sts_MaintByp : BOOL; {access Read Only}   // 1=A Maintenance Bypass is Active, display icon
   Sts_AlmInh : BOOL; {access Read Only}   // 1=An Alarm is Shelved, Disabled or Suppressed, display icon
   Sts_Err : BOOL; {access Read Only, visible}   // 1=Error in Config: see detail bits for reason
   Err_Timer : BOOL; {access Read Only}   // 1=Error in Config: Invalid Check Time (use 0 to 2147483)
   Err_Sim : BOOL; {access Read Only}   // 1=Error in Config: Invalid Simulation Time (use 0 to 2147483)
   Err_Alarm : BOOL; {access Read Only}   // 1=Error in Config: Alarm Min On Time, Shelf Time, Severity
   Sts_Hand : ALIAS FOR Mode.Sts_Hand; {access Read Only, visible}
   Sts_Maint : ALIAS FOR Mode.Sts_Maint; {access Read Only, visible}
   Sts_Ovrd : ALIAS FOR Mode.Sts_Ovrd; {access Read Only, visible}
   Sts_Prog : ALIAS FOR Mode.Sts_Prog; {access Read Only, visible}
   Sts_Oper : ALIAS FOR Mode.Sts_Oper; {access Read Only, visible}
   Sts_ProgOperLock : ALIAS FOR Mode.Sts_ProgOperLock; {access Read Only}
   Sts_NoMode : ALIAS FOR Mode.Sts_NoMode; {access Read Only}
   Sts_MAcqRcvd : ALIAS FOR Mode.Sts_MAcqRcvd; {access Read Only}
   Sts_FullStall : ALIAS FOR FullStall.Inp;   // 1=Valve Full Stall (failed to move at all)
   Alm_FullStall : ALIAS FOR FullStall.Alm;   // 1=Valve Full Stall (failed to move at all) Alarm
   Ack_FullStall : ALIAS FOR FullStall.Ack;   // 1=Full Stall Alarm has been acknowledged
   Sts_FullStallDisabled : ALIAS FOR FullStall.Disabled;   // 1=Full Stall Alarm has been Disabled by Maintenance
   Sts_FullStallShelved : ALIAS FOR FullStall.Shelved;   // 1=Full Stall Alarm has been Shelved by Operator
   Sts_FullStallSuppressed : ALIAS FOR FullStall.Suppressed;   // 1=Full Stall Alarm has been Suppressed by Program
   Sts_TransitStall : ALIAS FOR TransitStall.Inp;   // 1=Valve Transit Stall (did not reach target position)
   Alm_TransitStall : ALIAS FOR TransitStall.Alm;   // 1=Valve Transit Stall (did not reach target pos.) Alarm
   Ack_TransitStall : ALIAS FOR TransitStall.Ack;   // 1=Transit Stall Alarm has been acknowledged
   Sts_TransitStallDisabled : ALIAS FOR TransitStall.Disabled;   // 1=Transit Stall Alarm has been Disabled by Maintenance
   Sts_TransitStallShelved : ALIAS FOR TransitStall.Shelved;   // 1=Transit Stall Alarm has been Shelved by Operator
   Sts_TransitStallSuppressed : ALIAS FOR TransitStall.Suppressed;   // 1=Transit Stall Alarm has been Suppressed by Program
   Sts_IntlkTrip : ALIAS FOR IntlkTrip.Inp;   // 1=Valve de-energized by an Interlock NOT OK
   Alm_IntlkTrip : ALIAS FOR IntlkTrip.Alm;   // 1=Alarm: Valve de-energized by an Interlock NOT OK
   Ack_IntlkTrip : ALIAS FOR IntlkTrip.Ack;   // 1=Interlock Trip Alarm has been acknowledged
   Sts_IntlkTripDisabled : ALIAS FOR IntlkTrip.Disabled;   // 1=Interlock Trip Alarm has been Disabled by Maintenance
   Sts_IntlkTripShelved : ALIAS FOR IntlkTrip.Shelved;   // 1=Interlock Trip Alarm has been Shelved by Operator
   Sts_IntlkTripSuppressed : ALIAS FOR IntlkTrip.Suppressed;   // 1=Interlock Trip Alarm has been Suppressed Program
   Sts_IOFault : ALIAS FOR IOFault.Inp;   // I/O Comm Fault Status (0=OK, 1=Bad)
   Alm_IOFault : ALIAS FOR IOFault.Alm;   // 1=I/O Fault Alarm
   Ack_IOFault : ALIAS FOR IOFault.Ack;   // 1=I/O Fault Alarm has been acknowledged
   Sts_IOFaultDisabled : ALIAS FOR IOFault.Disabled;   // 1=I/O Fault Alarm has been Disabled by Maintenance
   Sts_IOFaultShelved : ALIAS FOR IOFault.Shelved;   // 1=I/O Fault Alarm has been Shelved by Operator
   Sts_IOFaultSuppressed : ALIAS FOR IOFault.Suppressed;   // 1=I/O Fault Alarm has been Suppressed by Program
   Rdy_Open : BOOL; {access Read Only}   // 1=Ready to receive OCmd_Open (enables HMI button)
   Rdy_Close : BOOL; {access Read Only}   // 1=Ready to receive OCmd_Close (enables HMI button)
   Rdy_Bypass : BOOL; {access Read Only}   // 1=Ready to receive OCmd_Bypass (enables HMI button)
   Rdy_Check : BOOL; {access Read Only}   // 1=Ready to receive OCmd_Check (enables HMI button)
   Rdy_Disable : BOOL; {access Read Only}   // 1=Ready to receive MCmd_Disable (enables HMI button)
   Rdy_Enable : BOOL; {access Read Only}   // 1=Ready to receive MCmd_Enable (enables HMI button)
   Rdy_Reset : BOOL; {access Read Only}   // 1=Ready to receive OCmd_Reset (enables HMI button)
   Rdy_ResetAckAll : BOOL; {access Read Only}   // 1=At least one Alarm or latched Shed condition requires Reset or Ack
   P_ValveSO : BOOL;   // Unique Parameter Name for auto - discovery
END_VAR
VAR
   Mode : P_Mode := (Cfg_PCmdClear := 1, Cfg_OvrdOverLock := 1, Rdy_OAcq := 1);   // Valve Mode Selection
   IOFault : P_Alarm := (Cfg_AckReqd := 1, Cfg_AllowShelve := 1, Cfg_AllowDisable := 1, Cfg_PCmdClear := 1, Cfg_Severity := 1000, Cfg_AlmMinOnT := 5, PCfg_AllowExist := 1, Ack := 1);   // I/O Fault Alarm
   IntlkTrip : P_Alarm := (Cfg_AckReqd := 1, Cfg_AllowShelve := 1, Cfg_AllowDisable := 1, Cfg_PCmdClear := 1, Cfg_Severity := 500, Cfg_AlmMinOnT := 5, PCfg_AllowExist := 1, Ack := 1);   // Interlock Trip Alarm
   TransitStall : P_Alarm := (Cfg_AckReqd := 1, Cfg_AllowShelve := 1, Cfg_AllowDisable := 1, Cfg_PCmdClear := 1, Cfg_Severity := 1000, Cfg_AlmMinOnT := 5, PCfg_AllowExist := 1, Ack := 1);   // Valve Transit Stall (moved but did not reach target) Alarm
   FullStall : P_Alarm := (Cfg_AckReqd := 1, Cfg_AllowShelve := 1, Cfg_AllowDisable := 1, Cfg_PCmdClear := 1, Cfg_Severity := 1000, Cfg_AlmMinOnT := 5, PCfg_AllowExist := 1, Ack := 1);   // Valve Full Stall (did not move) Alarm
   Cfg_Tag : STRING_20 := 'P_ValveSO';   // Tagname for display on HMI
   Cfg_Label : STRING_20 := 'Valve Control';   // Label for graphic symbol displayed on HMI
   Cfg_Desc : STRING_40 := 'Solenoid Operated Valve';   // Description for display on HMI
   Wrk_Open : BOOL; {access None}   // 1=Requested to OPEN Valve, 0=Requested to CLOSE Valve
   Wrk_SimOpenT : TIMER; {access None}   // Simulation Delay until Opened
   Wrk_SimCloseT : TIMER; {access None}   // Simulation Delay until Closed
   Wrk_OpenFdbk : BOOL; {access None}   // 1=LS Feedback shows valve confirmed open
   Wrk_Notify : DINT; {access None}   // Buffer for building Val_Notify
   Wrk_Bypass : BOOL; {access None}   // Internal Bypassable Permissives and Interlocks are Bypassed flag
   Wrk_Disabled : BOOL; {access None}   // Internal Valve is Disabled
   Wrk_ClosedFdbk : BOOL; {access None}   // 1=LS Feedback shows valve confirmed closed
   Wrk_TransitStallT : TIMER; {access Read Only}   // Timer for Transit Stall Check
   Wrk_FullStallT : TIMER; {access Read Only}   // Timer for Full Stall Check
   Inf_Tab : SINT;   // Tab to display (FTView ME)
   Wrk_Cmd : SINT; {access None}   // Buffer for building Val_Cmd
   Wrk_Sts : SINT; {access None}   // Buffer for building Val_Sts
   Wrk_Fault : SINT; {access None}   // Buffer for building Val_Fault
   Inf_Type : STRING_16 := 'P_ValveSO'; {access Read Only}   // Type identifier for HMI navigation
   Wrk_SimOpenLS : BOOL; {access None}   // Simulated valve Open Limit Switch
   Wrk_SimClosedLS : BOOL; {access None}   // Simulated valve Closed Limit Switch
   Inf_Lib : STRING_12 := 'RA-BAS'; {access Read Only}   // Display Library for Faceplate call-up
   Wrk_SrcQ : SINT; {access None}   // Register for building Source / Quality enumeration
   Wrk_NotRdy : BOOL; {access None}   // Device Not Ready conditions excluding shed latches
   Wrk_NoLongerSim : BOOL; {access None}   // Switched from Simulated to Real Valve this scan
END_VAR

ROUTINE EnableInFalse   (* ladder *)
// Disabled is asserted; Outputs OFF; Valve Status shown but Alarms disabled
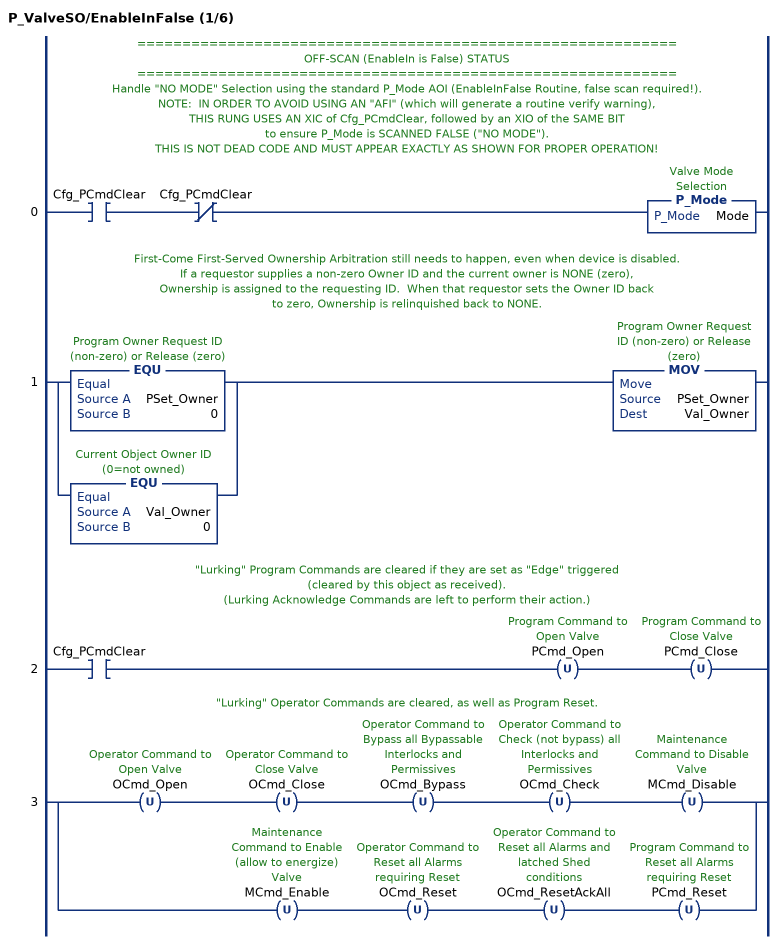
   // ============================================================
   // OFF-SCAN (EnableIn is False) STATUS
   // ============================================================
   // Handle "NO MODE" Selection using the standard P_Mode AOI (EnableInFalse Routine, false scan required!).
   // NOTE:  IN ORDER TO AVOID USING AN "AFI" (which will generate a routine verify warning),
   // THIS RUNG USES AN XIC of Cfg_PCmdClear, followed by an XIO of the SAME BIT
   // to ensure P_Mode is SCANNED FALSE ("NO MODE").
   // THIS IS NOT DEAD CODE AND MUST APPEAR EXACTLY AS SHOWN FOR PROPER OPERATION!
   0: XIC(Cfg_PCmdClear)XIO(Cfg_PCmdClear)P_Mode(Mode);
   // First-Come First-Served Ownership Arbitration still needs to happen, even when device is disabled.
   // If a requestor supplies a non-zero Owner ID and the current owner is NONE (zero),
   // Ownership is assigned to the requesting ID.  When that requestor sets the Owner ID back
   // to zero, Ownership is relinquished back to NONE.
   1: [EQU(PSet_Owner,0) ,EQU(Val_Owner,0) ]MOV(PSet_Owner,Val_Owner);
   // "Lurking" Program Commands are cleared if they are set as "Edge" triggered
   // (cleared by this object as received).
   // (Lurking Acknowledge Commands are left to perform their action.)
   2: XIC(Cfg_PCmdClear)OTU(PCmd_Open)OTU(PCmd_Close);
   // "Lurking" Operator Commands are cleared, as well as Program Reset.
   3: [OTU(OCmd_Open) OTU(OCmd_Close) OTU(OCmd_Bypass) OTU(OCmd_Check) OTU(MCmd_Disable) ,OTU(MCmd_Enable) OTU(OCmd_Reset) OTU(OCmd_ResetAckAll) OTU(PCmd_Reset) ];
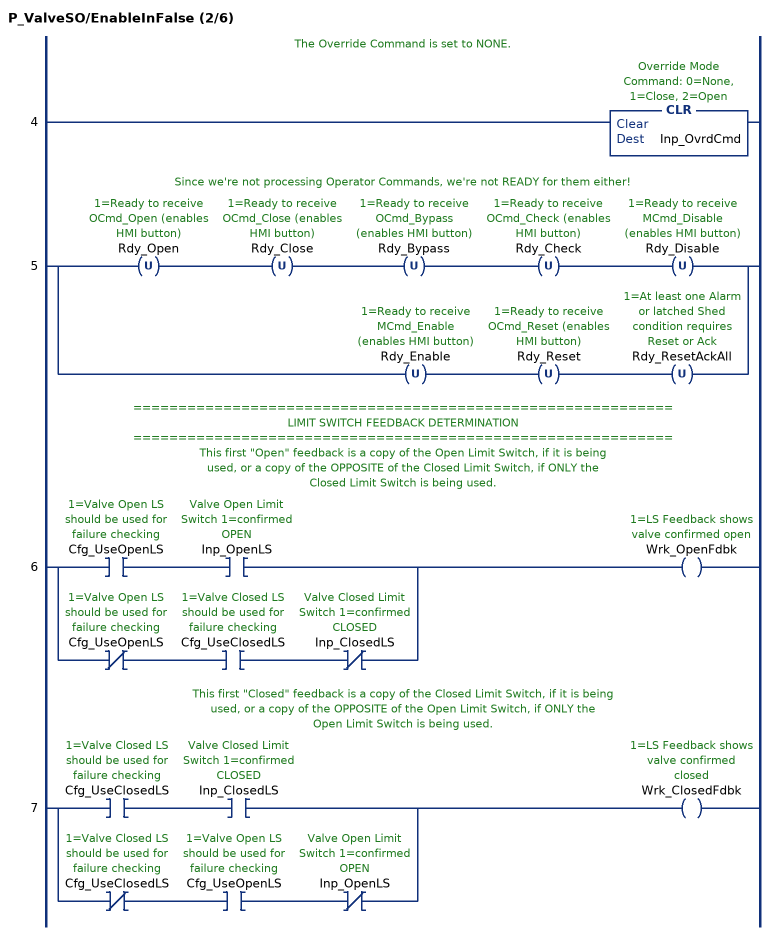
   // The Override Command is set to NONE.
   4: CLR(Inp_OvrdCmd);
   // Since we're not processing Operator Commands, we're not READY for them either!
   5: [OTU(Rdy_Open) OTU(Rdy_Close) OTU(Rdy_Bypass) OTU(Rdy_Check) OTU(Rdy_Disable) ,OTU(Rdy_Enable) OTU(Rdy_Reset) OTU(Rdy_ResetAckAll) ];
   // ============================================================
   // LIMIT SWITCH FEEDBACK DETERMINATION
   // ============================================================
   // This first "Open" feedback is a copy of the Open Limit Switch, if it is being
   // used, or a copy of the OPPOSITE of the Closed Limit Switch, if ONLY the
   // Closed Limit Switch is being used.
   6: [XIC(Cfg_UseOpenLS) XIC(Inp_OpenLS) ,XIO(Cfg_UseOpenLS) XIC(Cfg_UseClosedLS) XIO(Inp_ClosedLS) ]OTE(Wrk_OpenFdbk);
   // This first "Closed" feedback is a copy of the Closed Limit Switch, if it is being
   // used, or a copy of the OPPOSITE of the Open Limit Switch, if ONLY the
   // Open Limit Switch is being used.
   7: [XIC(Cfg_UseClosedLS) XIC(Inp_ClosedLS) ,XIO(Cfg_UseClosedLS) XIC(Cfg_UseOpenLS) XIO(Inp_OpenLS) ]OTE(Wrk_ClosedFdbk);
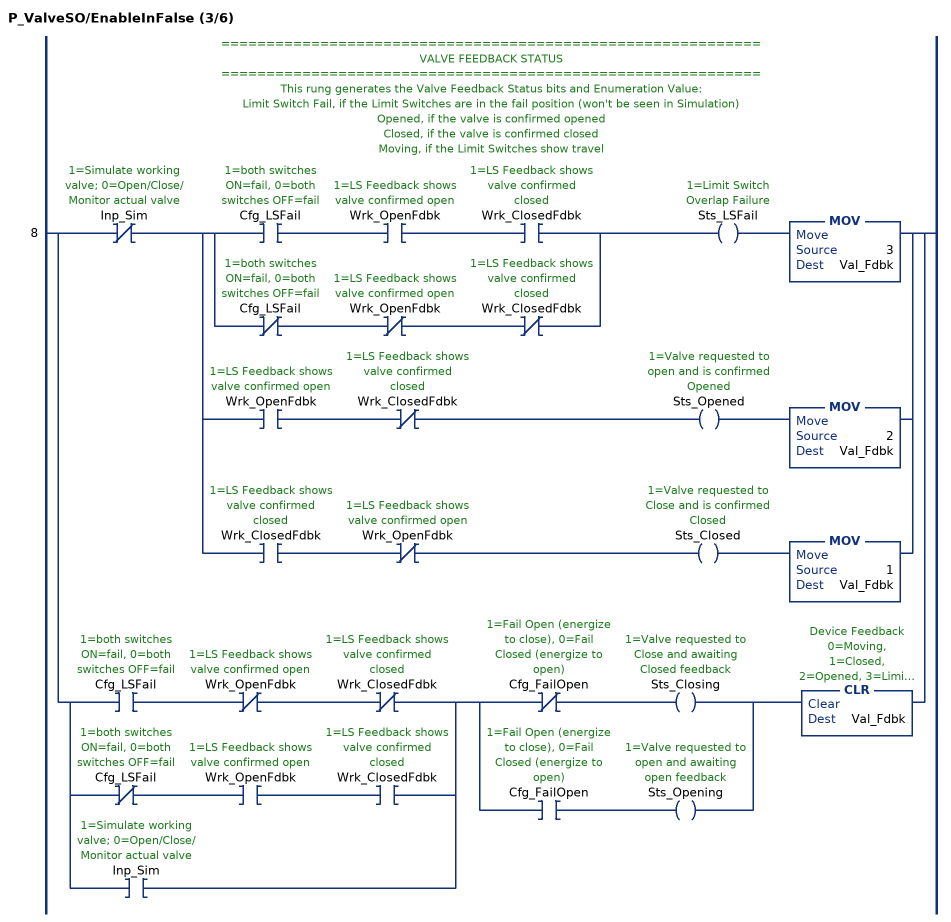
   // ============================================================
   // VALVE FEEDBACK STATUS
   // ============================================================
   // This rung generates the Valve Feedback Status bits and Enumeration Value:
   // Limit Switch Fail, if the Limit Switches are in the fail position (won't be seen in Simulation)
   // Opened, if the valve is confirmed opened
   // Closed, if the valve is confirmed closed
   // Moving, if the Limit Switches show travel
   8: [XIO(Inp_Sim) [[XIC(Cfg_LSFail) XIC(Wrk_OpenFdbk) XIC(Wrk_ClosedFdbk) ,XIO(Cfg_LSFail) XIO(Wrk_OpenFdbk) XIO(Wrk_ClosedFdbk) ] OTE(Sts_LSFail) MOV(3,Val_Fdbk) ,XIC(Wrk_OpenFdbk) XIO(Wrk_ClosedFdbk) OTE(Sts_Opened) MOV(2,Val_Fdbk) ,XIC(Wrk_ClosedFdbk) XIO(Wrk_OpenFdbk) OTE(Sts_Closed) MOV(1,Val_Fdbk) ] ,[[XIC(Cfg_LSFail) XIO(Wrk_OpenFdbk) XIO(Wrk_ClosedFdbk) ,XIO(Cfg_LSFail) XIC(Wrk_OpenFdbk) XIC(Wrk_ClosedFdbk) ] ,XIC(Inp_Sim) ] [XIO(Cfg_FailOpen) OTE(Sts_Closing) ,XIC(Cfg_FailOpen) OTE(Sts_Opening) ] CLR(Val_Fdbk) ];
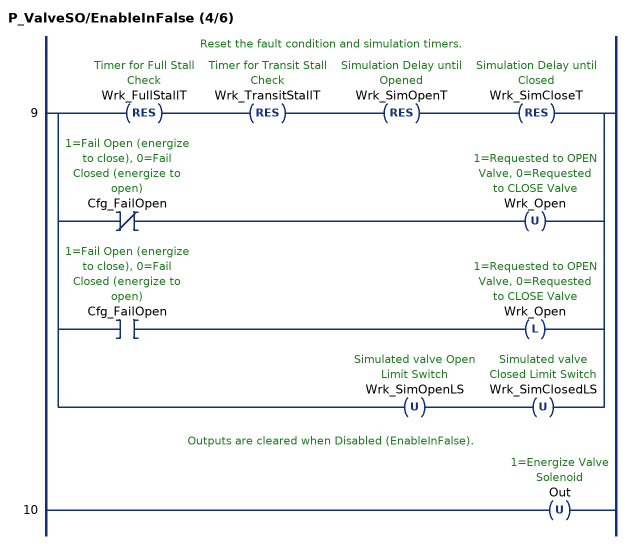
   // Reset the fault condition and simulation timers.
   9: [RES(Wrk_FullStallT) RES(Wrk_TransitStallT) RES(Wrk_SimOpenT) RES(Wrk_SimCloseT) ,[XIO(Cfg_FailOpen) OTU(Wrk_Open) ,XIC(Cfg_FailOpen) OTL(Wrk_Open) ] ,OTU(Wrk_SimOpenLS) OTU(Wrk_SimClosedLS) ];
   // Outputs are cleared when Disabled (EnableInFalse).
   10: OTU(Out);
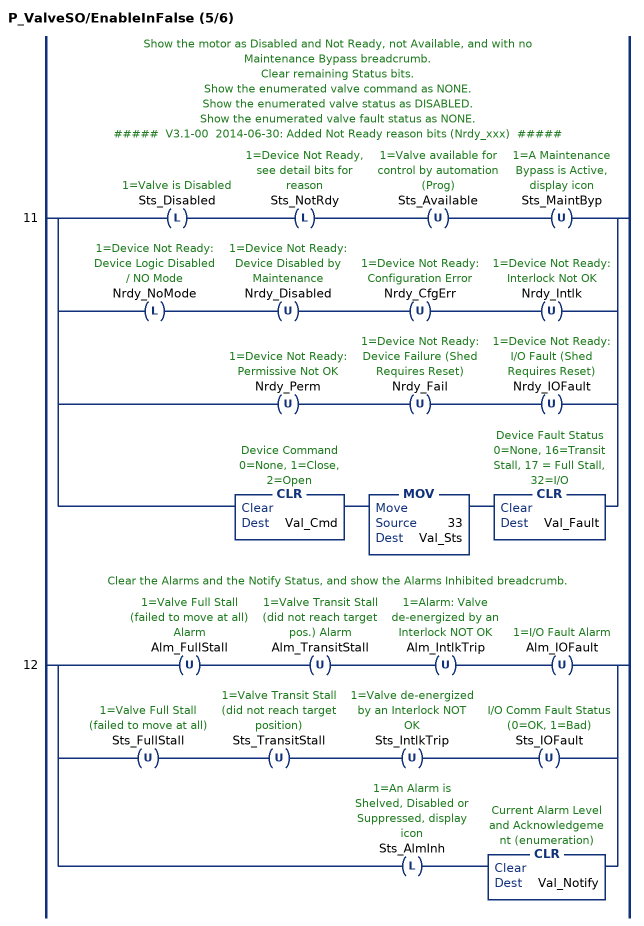
   // Show the motor as Disabled and Not Ready, not Available, and with no
   // Maintenance Bypass breadcrumb.
   // Clear remaining Status bits.
   // Show the enumerated valve command as NONE.
   // Show the enumerated valve status as DISABLED.
   // Show the enumerated valve fault status as NONE.
   // #####  V3.1-00  2014-06-30: Added Not Ready reason bits (Nrdy_xxx)  #####
   11: [OTL(Sts_Disabled) OTL(Sts_NotRdy) OTU(Sts_Available) OTU(Sts_MaintByp) ,OTL(Nrdy_NoMode) OTU(Nrdy_Disabled) OTU(Nrdy_CfgErr) OTU(Nrdy_Intlk) ,OTU(Nrdy_Perm) OTU(Nrdy_Fail) OTU(Nrdy_IOFault) ,CLR(Val_Cmd) MOV(33,Val_Sts) CLR(Val_Fault) ];
   // Clear the Alarms and the Notify Status, and show the Alarms Inhibited breadcrumb.
   12: [OTU(Alm_FullStall) OTU(Alm_TransitStall) OTU(Alm_IntlkTrip) OTU(Alm_IOFault) ,OTU(Sts_FullStall) OTU(Sts_TransitStall) OTU(Sts_IntlkTrip) OTU(Sts_IOFault) ,OTL(Sts_AlmInh) CLR(Val_Notify) ];
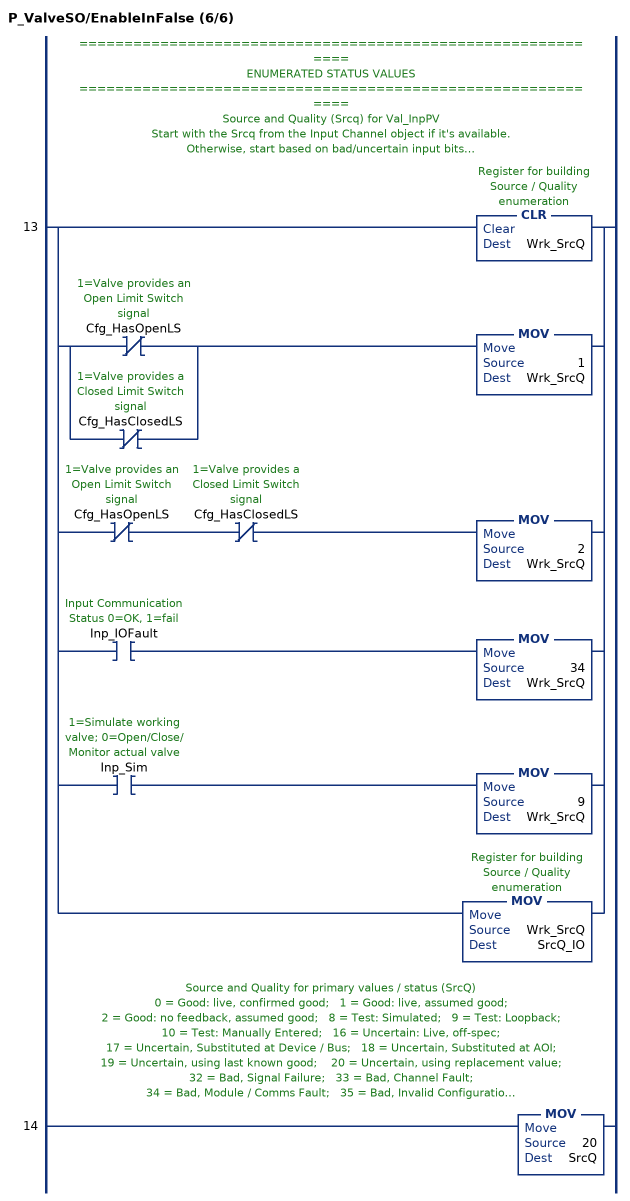
   // ============================================================
   // ENUMERATED STATUS VALUES
   // ============================================================
   // Source and Quality (Srcq) for Val_InpPV
   // Start with the Srcq from the Input Channel object if it's available.
   // Otherwise, start based on bad/uncertain input bits.
   // 0 = Good: live, confirmed good;   1 = Good: live, assumed good;
   // 2 = Good: no feedback, assumed good;   8 = Test: Simulated;   9 = Test: Loopback;
   // 10 = Test: Manually Entered;   16 = Uncertain: Live, off-spec;
   // 17 = Uncertain, Substituted at Device / Bus;   18 = Uncertain, Substituted at AOI;
   // 19 = Uncertain, using last known good;    20 = Uncertain, using replacement value;
   // 32 = Bad, Signal Failure;   33 = Bad, Channel Fault;
   // 34 = Bad, Module / Comms Fault;   35 = Bad, Invalid Configuration
   // #####  V3.1-00  2014-06-30:  Added rung for Source/Quality enumerations.  #####
   13: [CLR(Wrk_SrcQ) ,[XIO(Cfg_HasOpenLS) ,XIO(Cfg_HasClosedLS) ] MOV(1,Wrk_SrcQ) ,XIO(Cfg_HasOpenLS) XIO(Cfg_HasClosedLS) MOV(2,Wrk_SrcQ) ,XIC(Inp_IOFault) MOV(34,Wrk_SrcQ) ,XIC(Inp_Sim) MOV(9,Wrk_SrcQ) ,MOV(Wrk_SrcQ,SrcQ_IO) ];
   // Source and Quality for primary values / status (SrcQ)
   // 0 = Good: live, confirmed good;   1 = Good: live, assumed good;
   // 2 = Good: no feedback, assumed good;   8 = Test: Simulated;   9 = Test: Loopback;
   // 10 = Test: Manually Entered;   16 = Uncertain: Live, off-spec;
   // 17 = Uncertain, Substituted at Device / Bus;   18 = Uncertain, Substituted at AOI;
   // 19 = Uncertain, using last known good;    20 = Uncertain, using replacement value;
   // 32 = Bad, Signal Failure;   33 = Bad, Channel Fault;
   // 34 = Bad, Module / Comms Fault;   35 = Bad, Invalid Configuration
   // #####  V3.1-00  2014-06-30:  Added rung for Source/Quality enumerations.  #####
   14: MOV(20,SrcQ);
END_ROUTINE

ROUTINE Logic   (* ladder *)
// Normal Scan: control / monitor solenoid-operated valve
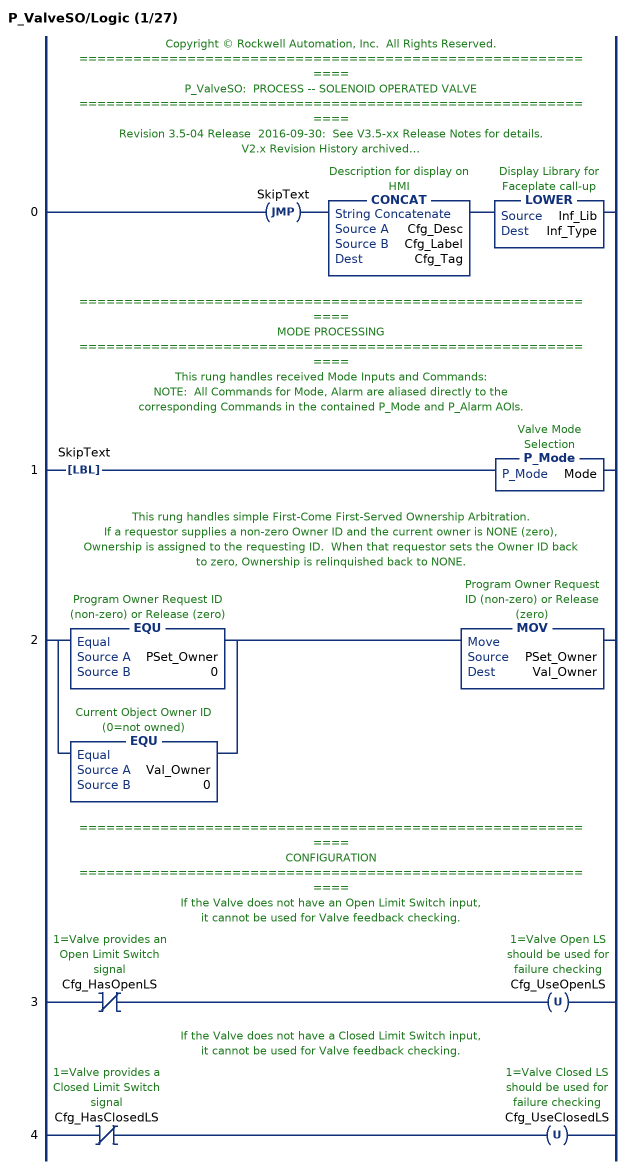
   // Copyright © Rockwell Automation, Inc.  All Rights Reserved.
   // ============================================================
   // P_ValveSO:  PROCESS -- SOLENOID OPERATED VALVE
   // ============================================================
   // Revision 3.5-04 Release  2016-09-30:  See V3.5-xx Release Notes for details.
   // V2.x Revision History archived.
   // V3.0-00  2013-06-30:  Added Inf_Lib. Using P_Alarm, P_Mode V3.0.
   // V3.0-01  2013-07-31:  Modified Parameter descriptions only.
   // V3.0-02  2013-09-03:  Modified Parameter descriptions only.
   // V3.0-03  2013-10-30:  Prescan code modified for proper powerup state.
   // Corrected Parameter descriptions and default
   // configuration values for alarms.
   // V3.0-04  2014-01-22:  Corrected Parameter Description for Val_Sts.
   // V3.1-00  2014-07-08:  Modified to use P_Alarm, P_Mode V3.1. Added Not
   // Ready reason bits (Nrdy_Xxxxx), source/quality values (SrcQ).
   // Modified to consistently use alias tag names.
   // V3.1-01  2014-09-03:  Exposed stall timers ACC/PRE (read-only). Corrections to
   // Nrdy_ trip and reset logic. Using P_Alarm, P_Mode V3.1-01.
   // V3.1-02  2014-09-30:  Unchanged, but using P_Alarm V3.1-02.
   // V3.5-01  2016-01-29:  Unchanged, but using P_Alarm V3.5.01.
   // V3.5-04  2016-09-30: Modified to align with actual device state on transition
   // from Sim to real valve.
   // ============================================================
   // This Instruction controls and monitors a single solenoid operated
   // valve (typ. two position: opened, closed) and provides:
   // *  Support for fail open (energize to close) and fail closed (energize to open, default) valves
   // *  Monitoring of limit switch feedback, display of actual valve status
   // *  Detection of failure to move (full stall), failure to reach position (transit stall)
   // *  Monitoring of Permissive conditions to allow energizing
   // *  Monitoring of Interlock conditions to de-energize
   // *  Simulation, providing feedback of a working valve while disabling outputs
   // *  Monitoring of I/O communication faults
   // *  Alarms for Full Stall, Transit Stall, Interlock Trip, I/O Fault
   // *  "Available" status for use by automation logic to know whether valve
   //       can be controlled by other objects.
   // Modes are provided by a P_Mode AOI instance.
   // Alarms are provided by P_Alarm AOI instances.
   // Modes of operation: Operator, Program, Override, Maintenance, Hand
   // ============================================================
   // SHOW LOCAL STRINGS
   // ============================================================
   // The STRINGs containing the text associated with each instance of this
   // instruction cannot be Input or Output Parameters, because STRINGs are not
   //  'atomic' types. (Inputs and Outputs must be SINT, INT, DINT, REAL, or BOOL.)
   // In order to make it easier to find and configure these STRINGs, this rung
   // was added.  THE JMP (and the LBL on the following rung)
   // MUST NOT BE REMOVED!!!
   // To view the STRINGs, go to the instruction instance (in LD or FBD), RIGHT-click
   // to bring up the context menu and select "Open Instruction Logic".
   // This rung will appear with the STRING values for the selected instance.
   // You may double-click the STRING values here to modify them as well.
   0: JMP(SkipText)CONCAT(Cfg_Desc,Cfg_Label,Cfg_Tag)LOWER(Inf_Lib,Inf_Type);
   // ============================================================
   // MODE PROCESSING
   // ============================================================
   // This rung handles received Mode Inputs and Commands:
   // NOTE:  All Commands for Mode, Alarm are aliased directly to the
   // corresponding Commands in the contained P_Mode and P_Alarm AOIs.
   1: LBL(SkipText)P_Mode(Mode);
   // This rung handles simple First-Come First-Served Ownership Arbitration.
   // If a requestor supplies a non-zero Owner ID and the current owner is NONE (zero),
   // Ownership is assigned to the requesting ID.  When that requestor sets the Owner ID back
   // to zero, Ownership is relinquished back to NONE.
   2: [EQU(PSet_Owner,0) ,EQU(Val_Owner,0) ]MOV(PSet_Owner,Val_Owner);
   // ============================================================
   // CONFIGURATION
   // ============================================================
   // If the Valve does not have an Open Limit Switch input,
   // it cannot be used for Valve feedback checking.
   3: XIO(Cfg_HasOpenLS)OTU(Cfg_UseOpenLS);
   // If the Valve does not have a Closed Limit Switch input,
   // it cannot be used for Valve feedback checking.
   4: XIO(Cfg_HasClosedLS)OTU(Cfg_UseClosedLS);
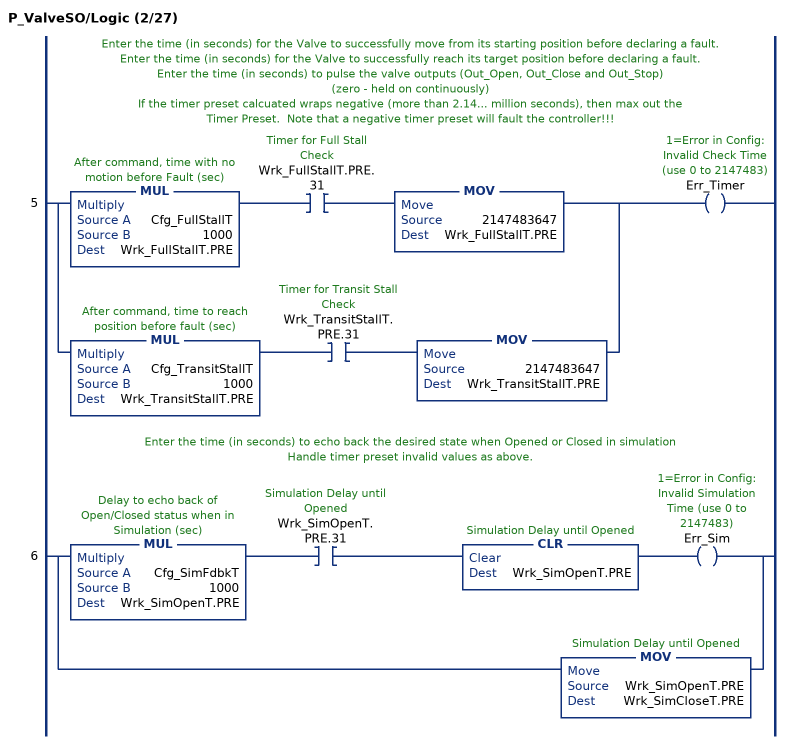
   // Enter the time (in seconds) for the Valve to successfully move from its starting position before declaring a fault.
   // Enter the time (in seconds) for the Valve to successfully reach its target position before declaring a fault.
   // Enter the time (in seconds) to pulse the valve outputs (Out_Open, Out_Close and Out_Stop)
   // (zero - held on continuously)
   // If the timer preset calcuated wraps negative (more than 2.14... million seconds), then max out the
   // Timer Preset.  Note that a negative timer preset will fault the controller!!!
   5: [MUL(Cfg_FullStallT,1000,Wrk_FullStallT.PRE) XIC(Wrk_FullStallT.PRE.31) MOV(2147483647,Wrk_FullStallT.PRE) ,MUL(Cfg_TransitStallT,1000,Wrk_TransitStallT.PRE) XIC(Wrk_TransitStallT.PRE.31) MOV(2147483647,Wrk_TransitStallT.PRE) ]OTE(Err_Timer);
   // Enter the time (in seconds) to echo back the desired state when Opened or Closed in simulation
   // Handle timer preset invalid values as above.
   6: [MUL(Cfg_SimFdbkT,1000,Wrk_SimOpenT.PRE) XIC(Wrk_SimOpenT.PRE.31) CLR(Wrk_SimOpenT.PRE) OTE(Err_Sim) ,MOV(Wrk_SimOpenT.PRE,Wrk_SimCloseT.PRE) ];
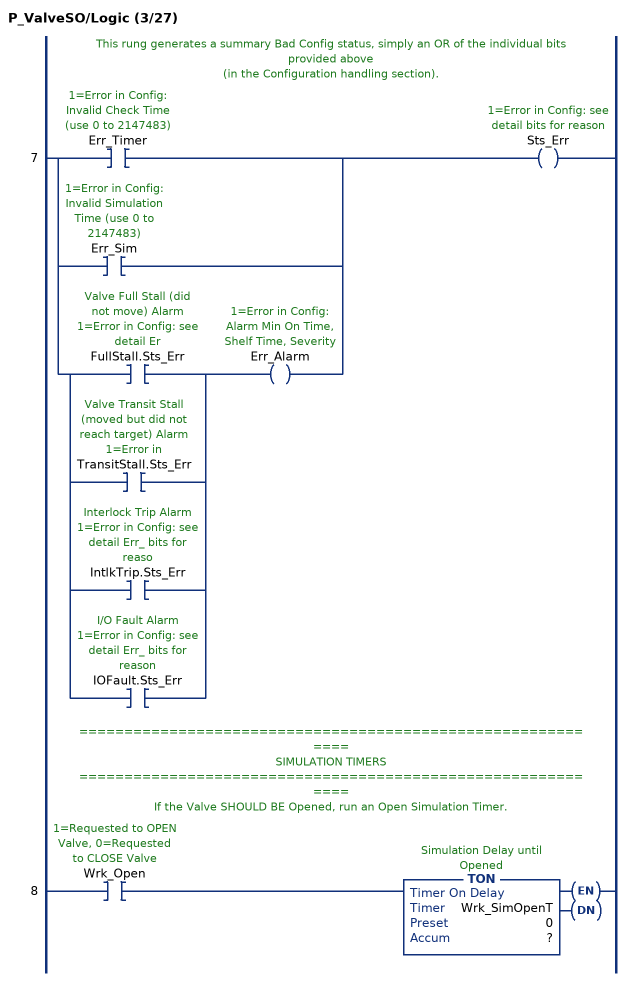
   // This rung generates a summary Bad Config status, simply an OR of the individual bits provided above
   // (in the Configuration handling section).
   7: [XIC(Err_Timer) ,XIC(Err_Sim) ,[XIC(FullStall.Sts_Err) ,XIC(TransitStall.Sts_Err) ,XIC(IntlkTrip.Sts_Err) ,XIC(IOFault.Sts_Err) ] OTE(Err_Alarm) ]OTE(Sts_Err);
   // ============================================================
   // SIMULATION TIMERS
   // ============================================================
   // If the Valve SHOULD BE Opened, run an Open Simulation Timer.
   8: XIC(Wrk_Open)TON(Wrk_SimOpenT,?,?);
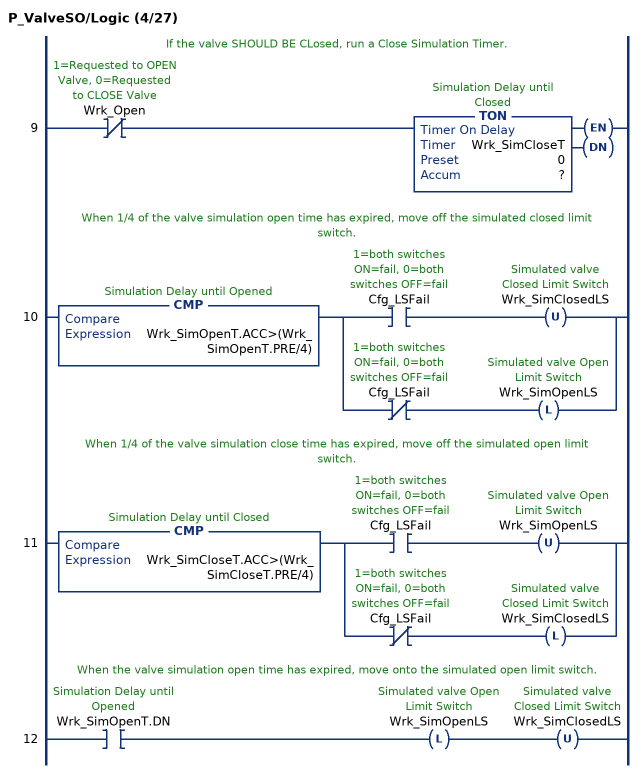
   // If the valve SHOULD BE CLosed, run a Close Simulation Timer.
   9: XIO(Wrk_Open)TON(Wrk_SimCloseT,?,?);
   // When 1/4 of the valve simulation open time has expired, move off the simulated closed limit switch.
   10: CMP(Wrk_SimOpenT.ACC>(Wrk_SimOpenT.PRE/4))[XIC(Cfg_LSFail) OTU(Wrk_SimClosedLS) ,XIO(Cfg_LSFail) OTL(Wrk_SimOpenLS) ];
   // When 1/4 of the valve simulation close time has expired, move off the simulated open limit switch.
   11: CMP(Wrk_SimCloseT.ACC>(Wrk_SimCloseT.PRE/4))[XIC(Cfg_LSFail) OTU(Wrk_SimOpenLS) ,XIO(Cfg_LSFail) OTL(Wrk_SimClosedLS) ];
   // When the valve simulation open time has expired, move onto the simulated open limit switch.
   12: XIC(Wrk_SimOpenT.DN)OTL(Wrk_SimOpenLS)OTU(Wrk_SimClosedLS);
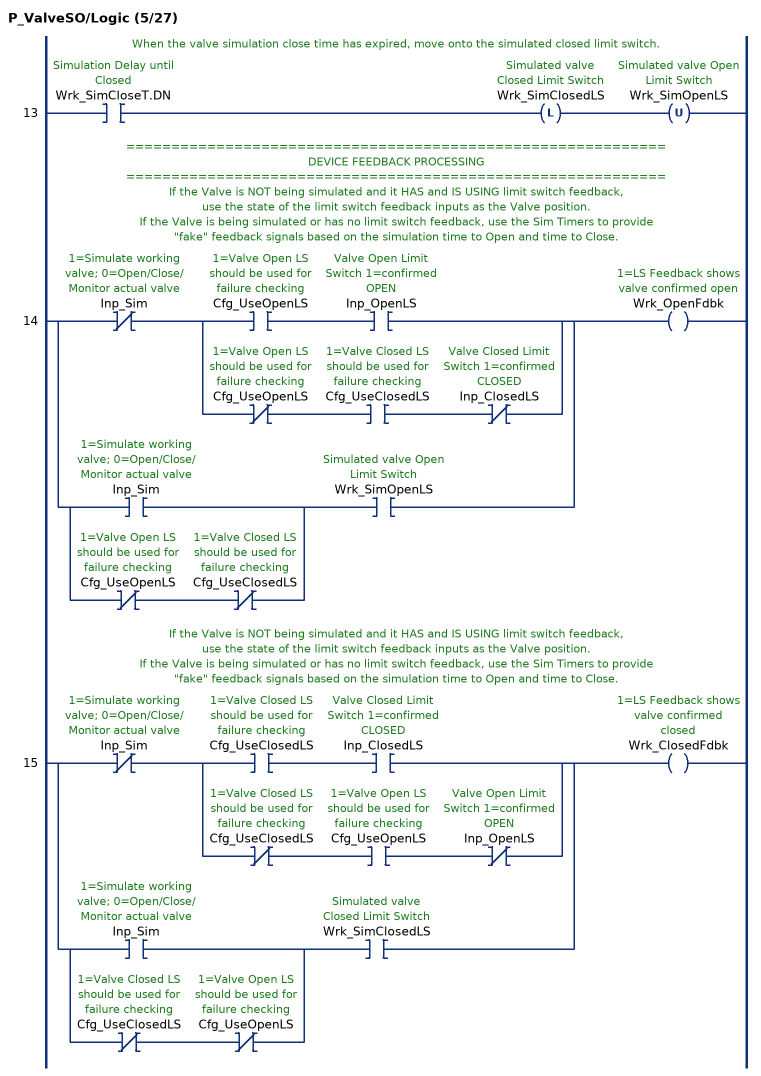
   // When the valve simulation close time has expired, move onto the simulated closed limit switch.
   13: XIC(Wrk_SimCloseT.DN)OTL(Wrk_SimClosedLS)OTU(Wrk_SimOpenLS);
   // ============================================================
   // DEVICE FEEDBACK PROCESSING
   // ============================================================
   // If the Valve is NOT being simulated and it HAS and IS USING limit switch feedback,
   // use the state of the limit switch feedback inputs as the Valve position.
   // If the Valve is being simulated or has no limit switch feedback, use the Sim Timers to provide
   // "fake" feedback signals based on the simulation time to Open and time to Close.
   14: [XIO(Inp_Sim) [XIC(Cfg_UseOpenLS) XIC(Inp_OpenLS) ,XIO(Cfg_UseOpenLS) XIC(Cfg_UseClosedLS) XIO(Inp_ClosedLS) ] ,[XIC(Inp_Sim) ,XIO(Cfg_UseOpenLS) XIO(Cfg_UseClosedLS) ] XIC(Wrk_SimOpenLS) ]OTE(Wrk_OpenFdbk);
   // If the Valve is NOT being simulated and it HAS and IS USING limit switch feedback,
   // use the state of the limit switch feedback inputs as the Valve position.
   // If the Valve is being simulated or has no limit switch feedback, use the Sim Timers to provide
   // "fake" feedback signals based on the simulation time to Open and time to Close.
   15: [XIO(Inp_Sim) [XIC(Cfg_UseClosedLS) XIC(Inp_ClosedLS) ,XIO(Cfg_UseClosedLS) XIC(Cfg_UseOpenLS) XIO(Inp_OpenLS) ] ,[XIC(Inp_Sim) ,XIO(Cfg_UseClosedLS) XIO(Cfg_UseOpenLS) ] XIC(Wrk_SimClosedLS) ]OTE(Wrk_ClosedFdbk);
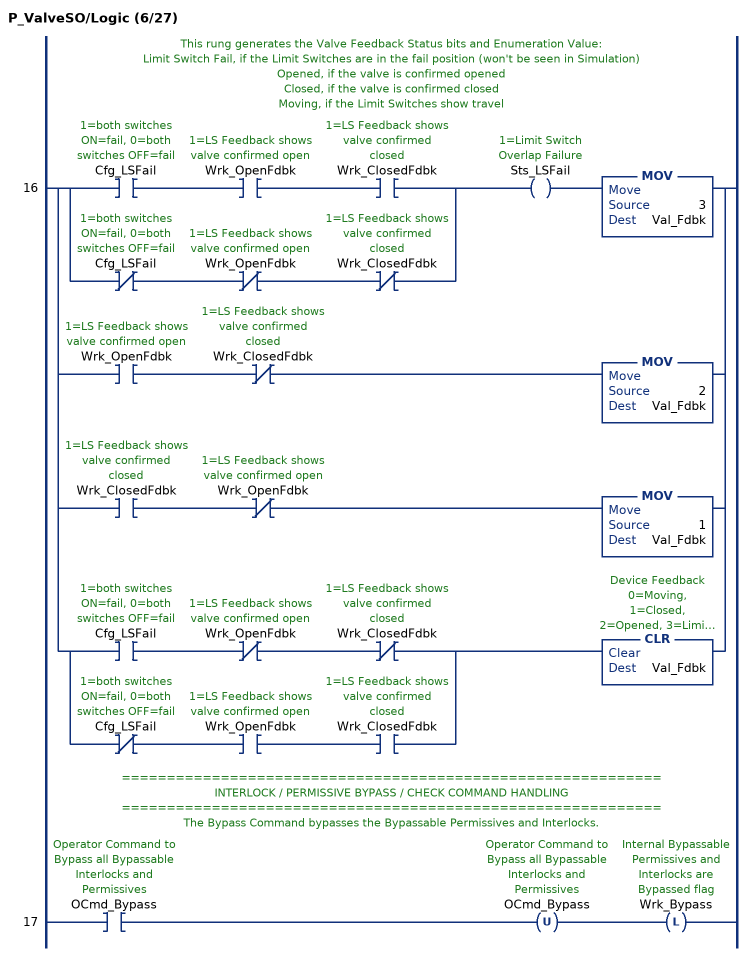
   // This rung generates the Valve Feedback Status bits and Enumeration Value:
   // Limit Switch Fail, if the Limit Switches are in the fail position (won't be seen in Simulation)
   // Opened, if the valve is confirmed opened
   // Closed, if the valve is confirmed closed
   // Moving, if the Limit Switches show travel
   16: [[XIC(Cfg_LSFail) XIC(Wrk_OpenFdbk) XIC(Wrk_ClosedFdbk) ,XIO(Cfg_LSFail) XIO(Wrk_OpenFdbk) XIO(Wrk_ClosedFdbk) ] OTE(Sts_LSFail) MOV(3,Val_Fdbk) ,XIC(Wrk_OpenFdbk) XIO(Wrk_ClosedFdbk) MOV(2,Val_Fdbk) ,XIC(Wrk_ClosedFdbk) XIO(Wrk_OpenFdbk) MOV(1,Val_Fdbk) ,[XIC(Cfg_LSFail) XIO(Wrk_OpenFdbk) XIO(Wrk_ClosedFdbk) ,XIO(Cfg_LSFail) XIC(Wrk_OpenFdbk) XIC(Wrk_ClosedFdbk) ] CLR(Val_Fdbk) ];
   // ============================================================
   // INTERLOCK / PERMISSIVE BYPASS / CHECK COMMAND HANDLING
   // ============================================================
   // The Bypass Command bypasses the Bypassable Permissives and Interlocks.
   17: XIC(OCmd_Bypass)OTU(OCmd_Bypass)OTL(Wrk_Bypass);
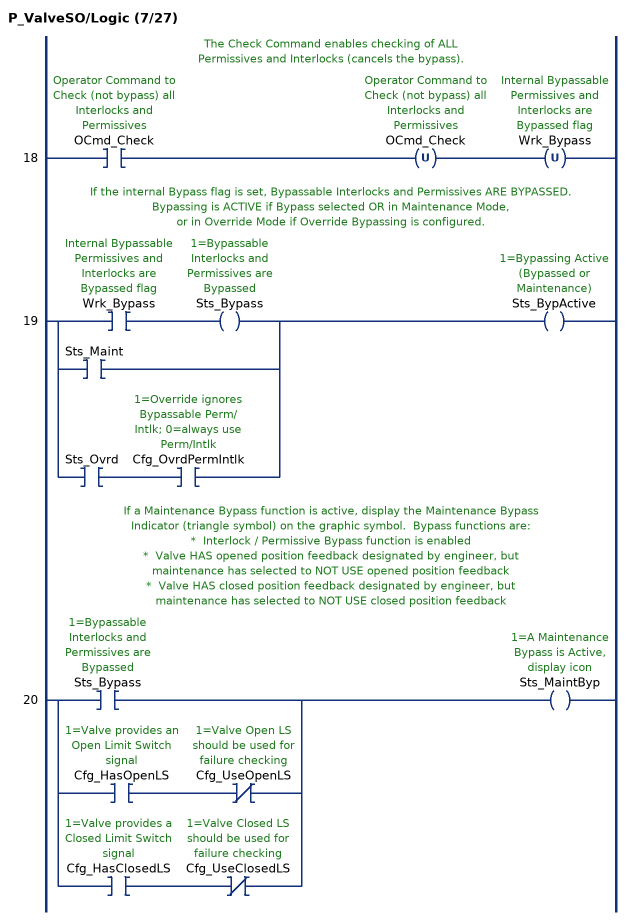
   // The Check Command enables checking of ALL
   // Permissives and Interlocks (cancels the bypass).
   18: XIC(OCmd_Check)OTU(OCmd_Check)OTU(Wrk_Bypass);
   // If the internal Bypass flag is set, Bypassable Interlocks and Permissives ARE BYPASSED.
   // Bypassing is ACTIVE if Bypass selected OR in Maintenance Mode,
   // or in Override Mode if Override Bypassing is configured.
   19: [XIC(Wrk_Bypass) OTE(Sts_Bypass) ,XIC(Sts_Maint) ,XIC(Sts_Ovrd) XIC(Cfg_OvrdPermIntlk) ]OTE(Sts_BypActive);
   // If a Maintenance Bypass function is active, display the Maintenance Bypass
   // Indicator (triangle symbol) on the graphic symbol.  Bypass functions are:
   // *  Interlock / Permissive Bypass function is enabled
   // *  Valve HAS opened position feedback designated by engineer, but
   // maintenance has selected to NOT USE opened position feedback
   // *  Valve HAS closed position feedback designated by engineer, but
   // maintenance has selected to NOT USE closed position feedback
   20: [XIC(Sts_Bypass) ,XIC(Cfg_HasOpenLS) XIO(Cfg_UseOpenLS) ,XIC(Cfg_HasClosedLS) XIO(Cfg_UseClosedLS) ]OTE(Sts_MaintByp);
